(* PLC project MQTT, CODESYS CODESYS V3.5 SP15 Patch 2, author Stefan Dreyer *)
(* stored: creationDateTime 2020-04-11T22:53:20.5572817, version 1.1.0.2, modificationDateTime 2020-04-11T22:45:00.0583058, organization Stefan Dreyer *)
(* MQTT Stuff
Using some cool stuff of OSCAT libs.
see oscat.de

more to describe *)

{attribute 'qualified_only'}
{attribute 'strict'}
TYPE ERRORS : (NOT_VALID := 0, CONNECTION_REFUSED := 1, MAX_PING_REPEATS := 2, RECEIVED_PUBISH_TO_BIG_FOR_BUFFER := 3, FULL_PACKET_NOT_RECEIVED := 4, RECEIVED_PUBLISH_REMAINING_LENGTH_ERROR := 5, NO_MORE_RECEIVE_SLOTS_FREE := 6, CONNECTION_ESTABLISHED := 7, TIMEOUT_CONNECTION := 8, REPEAT_PUBLISH_PUBCOMP := 9, REPEAT_PUBREL := 10, REORDER_PUBREC := 11, REORDER_PUBLISH_OUTGOING := 12, REPEAT_PUBLISH_PUBREC := 13, REPEAT_PUBLISH_PUBACK := 14, HARD_DISCONNECT := 15, MOVED_TO_BIG_RECEIVE_BUFFER := 16, NEED_BUFFER_MOV := 17, UNKNOWN_PAKET_RECEIVED := 18, TO_BIG_PAKET := 19, TOPIC_MOVED_DOWN := 20, TOPIC_AND_PAYLOAD_MOVED := 21, PAYLOAD_MOVED_UP := 22, TOPIC_MOVED_DOWN_NETWORK := 23, PAYLOAD_MOVED_UP_NETWORK := 24, REPEAT_PUBREC := 25, PUBEC_DISCHARGE := 26, REODER_PUBLISH_INCOMMING := 27, REORDER_PUBCOMP := 28, UNKNOWN_PAKET_IN_MQTT_IN_OUT := 29, PUBLISH_NO_SLOT_FREE := 30, OUT_OFF_DYN_MEMORY := 31);
END_TYPE

{attribute 'qualified_only'}
{attribute 'strict'}
TYPE INSERT_SPLIT_RETURN : (INSERT_NOT_VALID := 0, INSERT_DONE, INSERT_PENDING, INSERT_ERROR);
END_TYPE

TYPE MESSAGETYPE : (CONNECT := 16#10, CONNACK := 16#20, PUBLISH := 16#30, PUBACK := 16#40, PUBREC := 16#50, PUBREL := 16#60, PUBCOMP := 16#70, SUBSCRIBE := 16#80, SUBACK := 16#90, UNSUBSCRIBE := 16#A0, UNSUBACK := 16#B0, PINGREQ := 16#C0, PINGRESP := 16#D0, DISCONNECT := 16#E0) BYTE;
END_TYPE

{attribute 'qualified_only'}
{attribute 'strict'}
TYPE PROG_NUM : (Publish, Subscribe, ParseIncomming, MoveBuffer, ParsePublish, GetBufferFreePos, GetSplitTopic, DESTROY_HANDLE_MQTT, DESTROY_SPLIT_TOPIC, STATE_MASHINE_IN, STATE_MASHINE_OUT, SendOutData, SendInData, SendOutDataInsertTopic, SendOutDataInsertPayload, DESTROY_SPLIT_TOPIC_DONE, DESTROY_HANDLE_MQTT_DONE, DESTROY_CALLBACK_COLLECTOR, DESTROY_CALLBACK_COLLECTOR_DONE);
END_TYPE

{attribute 'qualified_only'}
{attribute 'strict'}
TYPE PUSHOVER_SOUND : (Standart := 1);
END_TYPE

TYPE QoS : (AtMostOnce := 2#0, AtLeastOnce := 2#1, ExactlyOnce := 2#10, Fail := 2#10000000) BYTE;
END_TYPE

{attribute 'qualified_only'}
{attribute 'strict'}
TYPE RECEIVE_TYPS : (FIND_PAYLOAD := 0, FIND_TOPIC := 1, FIND_LAST_TOPIC := 2, FIND_LAST_TOPIC_AND_PAYLOAD := 3);
END_TYPE

(* values of RECEIVER_INIT_TYPS: FIND_FULL_TOPIC: searching for full matching topic; FIND_LAST_TOPIC: searching for match of last topic; FIND_PAYLOAD: searching on paylod, from start, spared with delimiter; JSON_FULL: search full topic and one JSON element; JSON_SMALL: searching for last topic and one JSON element; MQTT_STRING: search with MQTT string(including +, #); MQTT_STRING_JSON: search with MQTT string(including +, #), then JSON *)

{attribute 'qualified_only'}
{attribute 'strict'}
TYPE RECEIVER_INIT_TYPS : (FIND_FULL_TOPIC := 0, FIND_LAST_TOPIC, FIND_PAYLOAD, JSON_FULL, JSON_SMALL, MQTT_STRING, MQTT_STRING_JSON);
END_TYPE

{attribute 'qualified_only'}
{attribute 'strict'}
TYPE STEPS_IN : (WAIT_DATA := 0, SEND_PUBACK, SEND_PUBREC, WAIT_PUBREL, SEND_PUBCOMP);
END_TYPE

{attribute 'qualified_only'}
{attribute 'strict'}
TYPE STEPS_OUT : (WAIT_DATA := 0, SEND_PUBLSIH, WAIT_PUBREC, SEND_PUBREL, WAIT_PUBCOMP, WAIT_PUBACK, WAIT_PINGRESP, SEND_SUBSCRIBE, WAIT_SUBACK, SEND_UNSUBSCRIBE, WAIT_UNSUBACK);
END_TYPE

{attribute 'qualified_only'}
{attribute 'strict'}
TYPE TOPIC_MATCH : (TOPIC_MATCHES := 1, TOPIC_DONT_MATCHES := 2, TOPIC_NO_MEMORY := 3) BYTE;
END_TYPE

{attribute 'qualified_only'}
{attribute 'strict'}
TYPE TOPIC_VALID : (TOPIC_UNTESTED := 0, TOPIC_VALID := 2, TOPIC_NOT_VALID := 1, TOPIC_NO_TEST := 3) BYTE;
END_TYPE

(* this data is passed to a subscription callback *)
TYPE CALLBACK_DATA : STRUCT
  PayloadString : POINTER TO STRING(255);  (* the Payload String, be aware, this pointer will only copy 255 bytes. If more needed, use memmove! *)
  Payload : POINTER TO BYTE;  (* pointer to binary payload *)
  PayloadSize : UDINT;  (* size of binary payload *)
  TopicOut : POINTER TO STRING(255);  (* here you get the compleete received topic string, maybe bigger then 255 byte! *)
  TopicOutSplit : POINTER TO SPLIT_TOPIC;  (* split topic.... *)
  PayloadIsString : BOOL;  (* Payload is string *)
END_STRUCT;
END_TYPE

{attribute 'enable_dynamic_creation'}
TYPE CALLBACK_INSTANCES : STRUCT
  callback : MQTT_SUBSCRIBE_CALLBACK;
  next : POINTER TO CALLBACK_INSTANCES := 0;
END_STRUCT;
END_TYPE

TYPE LIST_ALLVALUES_CALLBACK_DATA : STRUCT
  VarTYPE : CommonTypesAndFunctions.VAR_TYPES;
  Target : CommonTypesAndFunctions.ALL_TYPES_UNION_POINTER;
  SubTopic : POINTER TO STRING;  (* pointer to last subtopic or Payload Data to compare with *)
END_STRUCT;
END_TYPE

TYPE LIST_STRING_CALLBACK_DATA : STRUCT
  Target : POINTER TO STRING;  (* pointer to target string *)
  SubTopic : POINTER TO STRING;  (* pointer to last subtopic or Payload Data to compare with *)
END_STRUCT;
END_TYPE

TYPE MQTT_SUBSCRIBE_CALLBACKS : STRUCT
  Callback : MQTT_SUBSCRIBE_CALLBACK;
  ExpectingString : BOOL;  (* expecting string *)
  SplitTopic : POINTER TO HandleSplitTopic;
  free : BOOL := TRUE;  (* set to false if slot is aquired by an subscription *)
END_STRUCT;
END_TYPE

(* here the maximum sizes of paylod and topics are defined if dynamic low init of split topic is used, don't care about MaxTopicElementSize *)
TYPE COM_CONFIG : STRUCT
  MaxPayloadSize : UDINT := 2000;  (* max payload size *)
  MaxTopicLevels : UINT := 25;  (* max topic levels *)
  MaxTopicElementSize : UINT := 255;  (* Max Topic elemt size *)
END_STRUCT;
END_TYPE

TYPE DATA_FROM_BROKER : STRUCT
  MqttTopic : POINTER TO STRING;  (* use array in size of network buffer to split message dynamic, maybe not ... best is dynamic mammory.... or use an array of Pointer.... or callbacks so lets try to buffer public messages and releas one per cycle to application... now we try dynamic memmory.... MQTT Topic from Broker *)
  Topics : POINTER TO SPLIT_TOPIC;
  MqttPayload : POINTER TO BYTE;  (* MQTT Payload for Broker Payload from broker --> Pointer *)
  MqttPayloadSize : UDINT;  (* Payload size *)
  MessageType : MESSAGETYPE;  (* MQTT Message Type *)
  DataReceived : BOOL;  (* Data received *)
END_STRUCT;
END_TYPE

TYPE DATA_TO_BROKER : STRUCT
  PaketData : PAKET_DATA;  (* Data of Paket *)
END_STRUCT;
END_TYPE

(* contro struct between HANDLE_MQTT and MQTT_CONTROL *)
TYPE MQTT_COM : STRUCT
  S_BUF : NETWORK_BUFFER;
  R_BUF : NETWORK_BUFFER;
  MQTT_CON : BOOL;  (* if falling edge close with disconnect packet *)
  MQTT_ABORT : BOOL;  (* if using this to disconnect, don't send disconnect paket.... *)
  MQTT_URL : STRING(OSCAT_BASIC.STRING_LENGTH);
  MQTT_PACKET_NO : WORD;
  TIMEOUT : TIME;
  TLS : BOOL;  (* DNS_IP4 : DWORD; set to true if you want to use TLS *)
  TLS_CONFIG : POINTER TO CommonTypesAndFunctions.TLS_CONFIG := 0;  (* data to TLS stuff *)
  MQTT_RCV_STATE : BYTE;  (* 0= non 1= received 2= error *)
  ERROR_C : DWORD;
  ERROR_T : BYTE;
  CLIENT_ID : STRING(23);  (* CONNECT_TO_LOCALHOST:BOOL; *)
  CLIENT_WILL_TOPIC : STRING(255);  (* Topic vof will message after client id *)
  CLIENT_WILL_MESSAGE_DEAD : STRING(255);
  CLIENT_WILL_RETAIN : BOOL := TRUE;
  MQTT_NO_AWNSER : BOOL;  (* pakte wihout request-- return to receive state 1 *)
END_STRUCT;
END_TYPE

TYPE MQTT_IN_DATA : STRUCT
  step : STEPS_IN;
  PaketID : WORD;
  WaitsForBuffFree : ULINT;
  TimeOut : ton;
  TimeOutStarted : BOOL;
  PUBLISHOrder : UINT;
  PUBCOMPOrder : UINT;
  QoS : QoS;
  CountPubrecRepeat : UINT;
END_STRUCT;
END_TYPE

TYPE MQTT_IN_OUT : STRUCT
  handleFB : POINTER TO HANDLE_MQTT;  (* pointer to handle FB *)
  In : POINTER TO PAKET_DATA;
  InFree : BOOL := TRUE;  (* in free, true if free *)
  TDI : CommonTypesAndFunctions.TIME_DATE_IMPULS_DATA;  (* time, date, impulse... *)
  TLS_CONFIG : POINTER TO CommonTypesAndFunctions.TLS_CONFIG := 0;  (* TLS stuff data *)
  BROKER_CONNECTED : BOOL;
  COM_CONFIG : COM_CONFIG;  (* config for boot up *)
  ClientID : STRING(23) := 'CODESYS_MQTT';  (* client ID, only chars 0123456789abcdefghijklmnopqrstuvwxyzABCDEFGHIJKLMNOPQRSTUVWXYZ" System never can be anonymos *)
  BuildWillTopicAndMessage : BOOL := TRUE;
  WillTopicBase : STRING(255) := 'MQTTWill';
  ClientWillTopic : STRING(255) := 'DEAD';
  ClientWillMessage : STRING(30) := 'DIED';
  dynMemUsage : UDINT;  (* usage of dynamic RAM *)
  disconnectOnBufferOverflow : BOOL;  (* set this to one if you want the client to act like the standardt says if set to one and we receve mor publish pakets than we can handle, QoS 0 packets are lost and QoS 1 and 2 packets have to be repeaded by he broker *)
END_STRUCT;
END_TYPE

TYPE MQTT_INFO : STRUCT
  MQTT_CONNECTED : BOOL;
  MQTT_ERROR : STRING(OSCAT_BASIC.STRING_LENGTH);
END_STRUCT;
END_TYPE

TYPE MQTT_OUT_DATA : STRUCT
  InDataFromFb : POINTER TO PAKET_DATA;
  step : STEPS_OUT;
  WaitsForBuffFree : ULINT;
  PUBRECOrder : UINT;
  TimeOut : ton;
  TimeOutStarted : BOOL;
  PUBLISHOrder : UINT;
  PUBRELRepeatCounter : UINT;
END_STRUCT;
END_TYPE

TYPE ONE_ERROR : STRUCT
  error : ERRORS;
  when : DT;
  ERROR_C : DWORD;
  ERROR_T : BYTE;
  text : STRING(255);
END_STRUCT;
END_TYPE

TYPE PAKET_DATA : STRUCT
  MqttTopic : POINTER TO STRING;  (* MQTT Topic for Broker *)
  MqttTopicLength : UINT;  (* Topic length *)
  MqttPayload : POINTER TO BYTE;  (* MQTT Payload for Broker *)
  MqttPayloadLength : UDINT;  (* Payload length *)
  MessageType : MESSAGETYPE;  (* MQTT Message Type *)
  MessageQoS : QoS;  (* MQTT QoS *)
  SubackQoS : QoS;  (* SUCACK QoS Response *)
  MessageRetain : BOOL;  (* MQTT reatin *)
  DUP : BOOL;  (* Retry of paket *)
  PaketId : WORD;  (* PakatID for header *)
  SendSucsess : BOOL;  (* ID of MQTT FB to store or of request to Broker FbId:UINT; Send was succsessfull *)
  Callback : MQTT_SUBSCRIBE_CALLBACK;  (* Callback FB for subscription *)
  SplitTopic : POINTER TO HandleSplitTopic;  (* split topic for subscribe *)
  CallbackError : BOOL;  (* errore registering the callback *)
  ExpectingString : BOOL;  (* Expecting String *)
END_STRUCT;
END_TYPE

TYPE PUSHOVER_DATA : STRUCT
  Trigger : POINTER TO BOOL;
  Topic : POINTER TO STRING;
  Payload : POINTER TO STRING;
  Prio : USINT;
  Sound : PUSHOVER_SOUND;
  IsConfig : BOOL;
  R_T : R_TRIG;
  NeedToPush : BOOL;
  Negate : BOOL;
END_STRUCT;
END_TYPE

(* used for test cases... *)
TYPE RECEIVE_PAKET : STRUCT
  MqttTopic : STRING(2000);  (* MQTT Topic *)
  MqttPayload : STRING(2000);  (* MQTT Payload *)
END_STRUCT;
END_TYPE

TYPE REMAINING_LENGTH_RETURN : STRUCT
  RemainingLength : UDINT;
  IndexAfterRemainingLength : UINT;
  Error : BOOL;
  BuffToSmall : BOOL;  (* not all bytes of remaining length in buffer... *)
  SizeRemainingLength : USINT;  (* size of remaining length *)
END_STRUCT;
END_TYPE

TYPE SEND_INFOS : STRUCT
  SubscribeIndex : UINT;  (* this index is to be subscribed *)
  SubscribeNeeded : BOOL := FALSE;
  SubscribeBlocking : BOOL;
  UnsubscribeIndex : UINT;  (* this index is to be subscribed *)
  UnsubscribeNeeded : BOOL := FALSE;
  UnsubscribeBlocking : BOOL;
  PublishBlocking : BOOL;  (* this index is to be published *)
  PublishBlockingIndex : UINT;
  PingIndex : UINT;  (* this index is to be published *)
  PingNeeded : BOOL;
END_STRUCT;
END_TYPE

TYPE SPLIT_TOPIC : STRUCT
  Topics : POINTER TO POINTER TO STRING;  (* this is going to be a pointer to a array of pointer to stings *)
  ValidFields : UINT;  (* count of vailid fields in the array *)
END_STRUCT;
END_TYPE

{attribute 'qualified_only'}
VAR_GLOBAL CONSTANT  (* MyConstants *)
  QoS_BUFFER_SIZE : UINT := 50;
  NETWORK_BUFFER_LONG_SIZE : UINT := 4095;
  KEEP_ALIVE_TIME : DWORD := 8;
  SENDING_TIMEOUT : TIME := TIME#4s0ms;
  REPEAT_TIMEOUT : TIME := TIME#2s0ms;
  REORDER_VALUE : UINT := 50000;  (* 50000 *)
  SUBSTRACTION_VALUE : UINT := 30000;  (* 20000 *)
  MAX_PUBREL_REPEATS : UINT := 10;
END_VAR

{attribute 'qualified_only'}
VAR_GLOBAL  (* GVL_MQTT *)
  ProgNum : PROG_NUM;  (* Last Progamm stat for debug timeout exception *)
  LOG_BUFFER_MOVES : BOOL;
END_VAR

INTERFACE MQTT_SUBSCRIBE_CALLBACK
METHOD PublishReceived : BOOL
  VAR_INPUT
    Data : CALLBACK_DATA;  (* Collection of received Data *)
  END_VAR
END_METHOD
END_INTERFACE

PROGRAM Doku

            (*

Hello There,

with this library you are able to send and recvice MQTT paket on all QoS levels 0-2.

Use Pubish to publish data(Strings and binary),

Use subscribe to receive MQTT data. On Subscribe you can tell the FB if you are expecting an String as data, so you will get one on the pointer output.

How to use you can see in the example and testCase FB. This is my Test Case an it does up to 100 send and receives per second on an raspberry PI 1+ connectet to an mosquitto broker on an 
windows 10 maschine.

If you find errors, or anny instability, tell me, i will have a look.

TLS works fine without certificates.

This Projekt i using some parts of the grat OSCAT libs, so take a look at oscat.de

Greatings 

*)
          
END_PROGRAM

FUNCTION_BLOCK TestOutOfTheBoxNoTLS
  VAR_INPUT
    client : STRING := 'test.mosquitto.org:1883';  (* test.mosquitto.org *)
  END_VAR
  VAR
    MQTTClient : HANDLE_MQTT;
    MQTT_IN_OUT : MQTT_IN_OUT;
    publish : MQTTPublish;
    subscribe : MQTTSubscribe;
    ReceiveSubscribeTopic : STRING(255);
    ReceiveSubscribePayloadTick : STRING(255);
    ReceiveSubscribePayloadState : STRING(255);
    State : MQTTState;
    init : BOOL;
    varSend : BOOL;
    timerSend : ton;
    t1 : ton;
    t2 : ton;
    Payload : STRING;
    StringCallback : ListStringCallback;  (* the method PublishReceved() is call when an publsih packet form the broker is received. *)
    CallBackTargets : ARRAY[0..1] OF LIST_STRING_CALLBACK_DATA := [(Target := ADR(ReceiveSubscribePayloadState), SubTopic := ADR('State')), (Target := ADR(ReceiveSubscribePayloadTick), SubTopic := ADR('Tick'))];  (* the array contains the targets and sub topics for receive *)
  END_VAR

            //here init is done
IF NOT init THEN
	init := TRUE;
	MQTT_IN_OUT.ClientID := CONCAT('CodesysMqtt',TO_STRING(TICKS.GetTick(xDummy:= TRUE)));
	publish.SetMqttInOut(MQTT_IN_OUT:= ADR(MQTT_IN_OUT));
	subscribe.SetMqttInOut(MQTT_IN_OUT:= ADR(MQTT_IN_OUT));
	//init state FB, so you only have to call state();without parameters... 
	State.Init(
	State:= ADR(t1.Q), 
	Topic:= ADR('CODESYS-MQTT-BY-SD/State'), 
	StateName:= ADR(''), 
	StateValueOn:= ADR('On'), 
	StateValueOff:= ADR('Off'), 
	QoS:= QoS.ExactlyOnce, 
	RetainMqtt:= TRUE,
	MQTT_IN_OUT:= ADR(MQTT_IN_OUT));
	StringCallback.InitAsSplitTopic(ListData := ADR(CallBackTargets), LengthOfData:= 2);

END_IF
//timer for repeating packets
timerSend(in := NOT varSend, PT := T#2S);
varSend := timerSend.Q; 
t1(IN:= NOT t2.Q, PT:= T#1S, );
t2(IN:= t1.Q, PT:= T#1S, );
//call of MQTT client
MQTTClient( 
	MQTT_IN_OUT:= MQTT_IN_OUT, 
	ENABLE:= TRUE, 
	URL:= client, 
	TIMEOUT:= T#5S, 
	TLS:= FALSE);
//build payload
IF varSend THEN
	Payload:= TO_STRING(TICKS.GetTick(xDummy:= TRUE));
END_IF
//Publish Payload
publish(
	Topic:= ADR('CODESYS-MQTT-BY-SD/Tick'), 
	PayloadString:= ADR(Payload), 
	PublishAsString:= TRUE, 
	QoSIn:= QoS.ExactlyOnce, 
	MRetain:= TRUE, 
	send:= varSend);
//Subscribe to topic
subscribe(
	Subscribe:= TRUE, 
	Topic:= ADR('CODESYS-MQTT-BY-SD/#'), 
	QoSSubscribe:= QoS.ExactlyOnce, 
	ExpectingString:= TRUE,
	Callback:= StringCallback);


//call of state FB
State();
          
END_FUNCTION_BLOCK

FUNCTION_BLOCK TestOutOfTheBoxTLS
  VAR_INPUT
    client : STRING := 'test.mosquitto.org:8883';  (* test.mosquitto.org *)
  END_VAR
  VAR
    MQTTClient : HANDLE_MQTT;
    MQTT_IN_OUT : MQTT_IN_OUT;
    publish : MQTTPublish;
    subscribe : MQTTSubscribe;
    ReceiveSubscribeTopic : STRING(255);
    ReceiveSubscribePayloadTick : STRING(255);
    ReceiveSubscribePayloadState : STRING(255);
    State : MQTTState;
    init : BOOL;
    varSend : BOOL;
    timerSend : ton;
    t1 : ton;
    t2 : ton;
    Payload : STRING;
    StringCallback : ListStringCallback;  (* the method PublishReceved() is call when an publsih packet form the broker is received. *)
    CallBackTargets : ARRAY[0..1] OF LIST_STRING_CALLBACK_DATA := [(Target := ADR(ReceiveSubscribePayloadState), SubTopic := ADR('State')), (Target := ADR(ReceiveSubscribePayloadTick), SubTopic := ADR('Tick'))];  (* the array contains the targets and sub topics for receive *)
    TLS_CONFIG : CommonTypesAndFunctions.TLS_CONFIG;
  END_VAR

            //here init is done
IF NOT init THEN
	init := TRUE;
	MQTT_IN_OUT.ClientID := CONCAT('CodesysMqtt',TO_STRING(TICKS.GetTick(xDummy:= TRUE)));
	publish.SetMqttInOut(MQTT_IN_OUT:= ADR(MQTT_IN_OUT));
	subscribe.SetMqttInOut(MQTT_IN_OUT:= ADR(MQTT_IN_OUT));
	//init state FB, so you only have to call state();without parameters... 
	State.Init(
	State:= ADR(t1.Q), 
	Topic:= ADR('CODESYS-MQTT-BY-SD/State'), 
	StateName:= ADR(''), 
	StateValueOn:= ADR('On'), 
	StateValueOff:= ADR('Off'), 
	QoS:= QoS.ExactlyOnce, 
	RetainMqtt:= TRUE,
	MQTT_IN_OUT:= ADR(MQTT_IN_OUT));
	StringCallback.InitAsSplitTopic(ListData := ADR(CallBackTargets), LengthOfData:= 2);
	MQTT_IN_OUT.TLS_CONFIG := ADR(TLS_CONFIG);
END_IF
//timer for repeating packets
timerSend(in := NOT varSend, PT := T#2S);
varSend := timerSend.Q; 
t1(IN:= NOT t2.Q, PT:= T#1S, );
t2(IN:= t1.Q, PT:= T#1S, );
//call of MQTT client
MQTTClient( 
	MQTT_IN_OUT:= MQTT_IN_OUT, 
	ENABLE:= TRUE, 
	URL:= client, 
	TIMEOUT:= T#5S, 
	TLS:= TRUE);
//build payload
IF varSend THEN
	Payload:= TO_STRING(TICKS.GetTick(xDummy:= TRUE));
END_IF
//Publish Payload
publish(
	Topic:= ADR('CODESYS-MQTT-BY-SD/Tick'), 
	PayloadString:= ADR(Payload), 
	PublishAsString:= TRUE, 
	QoSIn:= QoS.ExactlyOnce, 
	MRetain:= TRUE, 
	send:= varSend);
//Subscribe to topic	
subscribe(
	Subscribe:= TRUE, 
	Topic:= ADR('CODESYS-MQTT-BY-SD/#'), 
	QoSSubscribe:= QoS.ExactlyOnce, 
	ExpectingString:= TRUE,
	Callback:= StringCallback);


//call of state FB
State();
          
END_FUNCTION_BLOCK

(* true if levels the same *)
FUNCTION CheckTopicLevel : BOOL
  VAR_INPUT
    s1 : POINTER TO STRING;  (* String from Broker *)
    s2 : POINTER TO STRING;  (* Subscribe String *)
  END_VAR
  VAR
    LenS1 : UINT;
  END_VAR

            CheckTopicLevel := FALSE;
//test Wildcard
IF (s2^[0] = CommonTypesAndFunctions.GetChar(in:= '+')) THEN //(s2[0] = GetChar(in:= '#')) OR  don't check # here
	CheckTopicLevel := TRUE;
	RETURN;	
END_IF
LenS1 := CommonTypesAndFunctions.len(STR:= s1); 
IF (LenS1 <> CommonTypesAndFunctions.len(STR:= s2)) THEN 
	RETURN;
END_IF//if len not eval then return
IF (CommonTypesAndFunctions.find(STR1:= s1, STR2:= s2) >= 0) OR (LenS1 = 0)THEN
	CheckTopicLevel := TRUE;
END_IF
          
END_FUNCTION

FUNCTION DoRemainingLength : USINT
  VAR_INPUT
    buffer : POINTER TO BYTE;
    RemainingLength : UINT;
  END_VAR
  VAR
    LocalLength : LINT;
    LocalBuffer : ARRAY[0..3] OF BYTE;
    BufferIndex : UINT := 0;
    TmpByte : BYTE;
  END_VAR

            //check if we have to move data for inserting remaining length
//borders are given in the mqtt doku
//
IF RemainingLength <= 128 THEN
	buffer[1] := UINT_TO_BYTE(RemainingLength);
	DoRemainingLength := 0;
ELSE
	LocalLength := RemainingLength;
	REPEAT
		TmpByte := LINT_TO_BYTE(LocalLength MOD 128);
		LocalLength := LocalLength / 128;
		IF LocalLength > 0 THEN
			TmpByte := TmpByte OR 128;
		END_IF
		LocalBuffer[BufferIndex] := TmpByte; 
		BufferIndex := BufferIndex +1;
	UNTIL 
		LocalLength <= 0 
	END_REPEAT
	//now move mem	
	//buffer index points to NEXT field, so sub 1
	MEM.MemMove(pSource:= buffer+2, pDestination:= buffer + 2 + BufferIndex - 1 , uiNumberOfBytes:= RemainingLength);
	CASE BufferIndex OF
		2: 	buffer[1]:= LocalBuffer[0];
			buffer[2]:= LocalBuffer[1];
			DoRemainingLength := 1;
		3:	buffer[1]:= LocalBuffer[0];
			buffer[2]:= LocalBuffer[1];
			buffer[3]:= LocalBuffer[2];
			DoRemainingLength := 2;
		4:	buffer[1]:= LocalBuffer[0];
			buffer[2]:= LocalBuffer[1];
			buffer[3]:= LocalBuffer[2];
			buffer[4]:= LocalBuffer[3];
			DoRemainingLength := 3;
		
	END_CASE
	
END_IF

          
END_FUNCTION

(* here no move of data, call remainig length bevor moving topic and paylod, use this for borders are given in the mqtt doku use this for publish pakets *)
FUNCTION DoRemainingLengthBevor : USINT
  VAR_INPUT
    buffer : POINTER TO BYTE;  (* points to start of buffer, not to start of remainig length! *)
    SizeTopic : UDINT;
    SizePayload : UDINT;
    InQoS : QoS;
  END_VAR
  VAR
    RemainingLength : UDINT;
    LocalLength : LINT;
    LocalBuffer : ARRAY[0..3] OF BYTE;
    BufferIndex : UINT := 0;
    TmpByte : BYTE;
  END_VAR

            
	
RemainingLength := SizeTopic + SizePayload;
	
RemainingLength := RemainingLength + 2;//add topic size encoding space
IF NOT (InQoS = QoS.AtMostOnce) THEN
	RemainingLength := RemainingLength + 2;//add space for paket identifier
END_IF

IF RemainingLength <= 128 THEN
	buffer[1] := UDINT_TO_BYTE(RemainingLength);
	DoRemainingLengthBevor := 0;
ELSE
	LocalLength := RemainingLength;
	REPEAT
		TmpByte := LINT_TO_BYTE(LocalLength MOD 128);
		LocalLength := LocalLength / 128;
		IF LocalLength > 0 THEN
			TmpByte := TmpByte OR 128;
		END_IF
		LocalBuffer[BufferIndex] := TmpByte; 
		BufferIndex := BufferIndex +1;
	UNTIL 
		LocalLength <= 0 
	END_REPEAT
	CASE BufferIndex OF
		2: 	buffer[1]:= LocalBuffer[0];
			buffer[2]:= LocalBuffer[1];
			DoRemainingLengthBevor := 1;
		3:	buffer[1]:= LocalBuffer[0];
			buffer[2]:= LocalBuffer[1];
			buffer[3]:= LocalBuffer[2];
			DoRemainingLengthBevor := 2;
		4:	buffer[1]:= LocalBuffer[0];
			buffer[2]:= LocalBuffer[1];
			buffer[3]:= LocalBuffer[2];
			buffer[4]:= LocalBuffer[3];
			DoRemainingLengthBevor := 3;
		
	END_CASE
	
END_IF

          
END_FUNCTION

FUNCTION GetRemainingLength : REMAINING_LENGTH_RETURN
  VAR_INPUT
    Buff : POINTER TO BYTE;  (* Pointer to Buffer *)
    pos : UINT;  (* Start of data in Buffer *)
    BuffSize : UDINT;
  END_VAR
  VAR
    BufferIndex : UINT := 1;
    Multipler : UDINT := 1;
    TmpByte : BYTE;
  END_VAR

            GetRemainingLength.Error := FALSE;
GetRemainingLength.SizeRemainingLength:= 0;

GetRemainingLength.BuffToSmall := FALSE;
BufferIndex := pos + 1;
REPEAT
	IF BufferIndex > (BuffSize - 1) THEN
		GetRemainingLength.BuffToSmall := TRUE;
	ELSE
		TmpByte := Buff[BufferIndex];
		BufferIndex := BufferIndex + 1;
		GetRemainingLength.RemainingLength := GetRemainingLength.RemainingLength + (TmpByte AND 127) * Multipler;
		Multipler := Multipler *128;
		IF Multipler > 128*128*128 THEN
			GetRemainingLength.RemainingLength := 0;//lengt 0 if broken
			GetRemainingLength.Error := TRUE;
		END_IF
	END_IF
	GetRemainingLength.SizeRemainingLength := GetRemainingLength.SizeRemainingLength + 1;
UNTIL
	TmpByte.7 = FALSE OR GetRemainingLength.BuffToSmall
	//TmpByte.7 = FALSE  OR GetRemainingLength.RemainingLength = 0 OR GetRemainingLength.BuffToSmall
END_REPEAT
GetRemainingLength.IndexAfterRemainingLength := BufferIndex;
          
END_FUNCTION

FUNCTION InitMQTTValue : BOOL
  VAR_INPUT
    DataArray : POINTER TO CommonTypesAndFunctions.PWConfigs;
    CountOfArray : UINT;
    ValueToMQTTArray : POINTER TO MQTTValue;
    MQTT_IN_OUT : POINTER TO MQTT_IN_OUT;
  END_VAR
  VAR
    i : UINT;
  END_VAR

            FOR i := 0 TO CountOfArray - 1 DO
	IF DataArray[i].NeedsMQTT THEN
		ValueToMQTTArray[i].Init(
			Topic:= DataArray[i].MQTTTopic, 
			ValueName:= DataArray[i].MQTTName, 
			ValuePointer:= DataArray[i].PointerTo, 
			ValueType:= DataArray[i].ValueType, 
			ValueDiff:= DataArray[i].MQTTDiff, 
			DecimalPlace:= DataArray[i].MQTTDezimal, 
			QoS:= DataArray[i].MQTTQoS, 
			RetainMqtt:= DataArray[i].MQTTRetain, 
			MinTime:= DataArray[i].MQTTTime,
			MQTT_IN_OUT:= MQTT_IN_OUT);
	END_IF
END_FOR
          
END_FUNCTION

(* returnds new pos in buff *)
FUNCTION InsertStringToBufferAndLength : UINT
  VAR_INPUT
    Str : POINTER TO STRING;
    buff : POINTER TO BYTE;  (* address to buffer *)
    pos : UINT;  (* Start to insert *)
  END_VAR
  VAR
    length : UINT;
  END_VAR

            length := CommonTypesAndFunctions.LEN(Str);
buff[pos]:= OSCAT_BASIC.BYTE_OF_DWORD(in:= length, N:= 1);
buff[pos+1]:= OSCAT_BASIC.BYTE_OF_DWORD(in:= length, N:= 0);

MEM.MemMove(pSource:= str, pDestination:= ADR(buff[pos+2]), uiNumberOfBytes:= length);
InsertStringToBufferAndLength := pos + length + 2;
          
END_FUNCTION

(* this FB collects instances of FB with the MQTT_SUBSCRIBE_CALLBACK interface. then you can pass a instance of this FB to a subscription FB to call all of your FBs to a specific subscription topic, in this call you can check if the packet was for your instance. If your instance methode call return true, the the FB exits the loop an so you may save cycle time. MEmory for instance references are created dynamic, so no restriction by library *)
FUNCTION_BLOCK CallbackCollector IMPLEMENTS MQTT_SUBSCRIBE_CALLBACK
  VAR
    first : POINTER TO CALLBACK_INSTANCES := 0;
    items : UDINT;
    size : UDINT;
  END_VAR

            
          

(* true if all ok, else false *)
METHOD put : BOOL
  VAR_INPUT
    instance : MQTT_SUBSCRIBE_CALLBACK;
  END_VAR
  VAR
    aktElement : POINTER TO CALLBACK_INSTANCES;
  END_VAR
                  aktElement := first;

IF aktElement = 0 THEN
	//first hit...
	{info 'semaphore'}
	first := __NEW(CALLBACK_INSTANCES);
	IF first = 0 THEN
		put := FALSE;
		RETURN;
	END_IF
	aktElement := first;
ELSE
	//search last
	WHILE aktElement^.next  <> 0 DO 
		aktElement := aktElement^.next; 
	END_WHILE
	{info 'semaphore'}
	aktElement^.next := __NEW(CALLBACK_INSTANCES);
	IF aktElement^.next = 0 THEN
		put := FALSE;
		RETURN;
	END_IF
	aktElement := aktElement^.next;
END_IF

aktElement^.callback := instance;
put := TRUE;
items := items + 1;
size := size + SIZEOF(CALLBACK_INSTANCES);
                
END_METHOD

METHOD PublishReceived : BOOL
  VAR_INPUT
    Data : CALLBACK_DATA;  (* Collection of received Data *)
  END_VAR
  VAR
    element : POINTER TO CALLBACK_INSTANCES;
    loop : BOOL := TRUE;
  END_VAR
                  

IF first = 0 THEN
	//no callback avalable
	RETURN;
END_IF
element := first;


WHILE loop DO
	IF element^.callback.PublishReceived(Data := Data) THEN
		PublishReceived := TRUE;
		RETURN;
	END_IF
	IF element^.next = 0 THEN
		loop := FALSE;
	ELSE
		element := element^.next;
	END_IF
END_WHILE

                
END_METHOD

(* destroy all dynamic content *)
METHOD destroy : BOOL
  VAR
    aktElement : POINTER TO CALLBACK_INSTANCES;
    nextElement : POINTER TO CALLBACK_INSTANCES;
  END_VAR
                  GVL_MQTT.ProgNum := PROG_NUM.DESTROY_CALLBACK_COLLECTOR;
IF first = 0 THEN
	RETURN;
END_IF

aktElement := first;

REPEAT
	nextElement := aktElement^.next;
	__DELETE(aktElement);
	aktElement := nextElement;
	items := items - 1;
	size := size - SIZEOF(CALLBACK_INSTANCES);
UNTIL aktElement = 0
END_REPEAT
first := 0;
GVL_MQTT.ProgNum := PROG_NUM.DESTROY_CALLBACK_COLLECTOR_DONE;
                
END_METHOD

METHOD FB_Exit : BOOL
  VAR_INPUT
    bInCopyCode : BOOL;  (* TRUE: the exit method is called in order to leave the instance which will be copied afterwards (online change). *)
  END_VAR
                  destroy();
                
END_METHOD
END_FUNCTION_BLOCK

FUNCTION_BLOCK ReceiverBase
  VAR
    MatchTyp : RECEIVER_INIT_TYPS;
    Target : CommonTypesAndFunctions.ALL_TYPES_UNION_POINTER;
    TargetType : CommonTypesAndFunctions.VAR_TYPES;
    PayloadCompare : POINTER TO STRING;
    TopicCompare : POINTER TO STRING;
    delimiter : BYTE;
    delimiterString : STRING(3);
    SplitTopic : HandleSplitTopic;
  END_VAR

            
          

METHOD init
  VAR_INPUT
    MQTT_IN_OUT : POINTER TO MQTT_IN_OUT;
    MatchTyp : RECEIVER_INIT_TYPS;
    Target : CommonTypesAndFunctions.ALL_TYPES_UNION_POINTER;
    TargetType : CommonTypesAndFunctions.VAR_TYPES;
    PayloadCompare : POINTER TO STRING;
    TopicCompare : POINTER TO STRING;
    delimiter : BYTE;
  END_VAR
                  MatchTyp := MatchTyp;
Target := Target;
TargetType := TargetType;
PayloadCompare := PayloadCompare;
TopicCompare := TopicCompare;
delimiter := delimiter;
delimiterString[0] := delimiter;
delimiterString[1] := 0;

IF MatchTyp = RECEIVER_INIT_TYPS.MQTT_STRING or MatchTyp = RECEIVER_INIT_TYPS.MQTT_STRING_JSON THEN
	SplitTopic.LowInit(TopicsLevelInit:= MQTT_IN_OUT^.COM_CONFIG.MaxTopicLevels,
			 SplitElementSizeInit:= MQTT_IN_OUT^.COM_CONFIG.MaxTopicElementSize, dynMemUsageInit:= ADR(MQTT_IN_OUT^.dynMemUsage));
	SplitTopic.NewTopic(in:= TopicCompare, test:= TRUE, SizeOfString:= CommonTypesAndFunctions.len(str:= TopicCompare));
END_IF
                
END_METHOD

METHOD CheckMatch : BOOL
  VAR_INPUT
    Data : CALLBACK_DATA;  (* Collection of received Data *)
  END_VAR
  VAR
    foundPos : DINT;
  END_VAR
                  CheckMatch := FALSE;
CASE MatchTyp OF
	RECEIVER_INIT_TYPS.FIND_FULL_TOPIC:
		IF CommonTypesAndFunctions.StrEquals(str1:= Data.TopicOut , str2:= PayloadCompare) THEN
			CheckMatch := TRUE;
			GetValue(fromWhere:= Data.PayloadString);
			RETURN;
		END_IF 
	RECEIVER_INIT_TYPS.FIND_LAST_TOPIC:
		IF CommonTypesAndFunctions.StrEquals(str1:= Data.TopicOutSplit^.Topics[Data.TopicOutSplit^.ValidFields - 1], str2:= PayloadCompare) THEN
			CheckMatch := TRUE;
			GetValue(fromWhere:= Data.PayloadString);
			RETURN;
		END_IF
	RECEIVER_INIT_TYPS.FIND_PAYLOAD:
		IF CommonTypesAndFunctions.StrEqualsAtStartWithDelimiter(str1:= PayloadCompare, str2:= Data.PayloadString , delimiter:= delimiter) THEN
			CheckMatch := TRUE;
			GetValue(fromWhere:= Data.PayloadString + TO_UINT(CommonTypesAndFunctions.find(str1:= Data.PayloadString, str2:= ADR(delimiterString)))+1);
			RETURN;	
		END_IF
	RECEIVER_INIT_TYPS.JSON_FULL:
		IF CommonTypesAndFunctions.StrEquals(str1:= Data.TopicOut , str2:= PayloadCompare) THEN
			foundPos := CommonTypesAndFunctions.find(str1:= Data.PayloadString, str2:= TopicCompare); 
			IF foundPos >= 0 THEN
				CheckMatch := TRUE;
				RETURN;	
			END_IF
		END_IF
	RECEIVER_INIT_TYPS.JSON_SMALL:
		IF CommonTypesAndFunctions.StrEquals(str1:= Data.TopicOutSplit^.Topics[Data.TopicOutSplit^.ValidFields - 1], str2:= PayloadCompare) THEN
			IF CommonTypesAndFunctions.find(str1:= Data.PayloadString, str2:= TopicCompare) >= 0 THEN
				CheckMatch := TRUE;
				RETURN;	
			END_IF
		END_IF
	RECEIVER_INIT_TYPS.MQTT_STRING:
		IF SplitTopic.CheckTopicMatchToMe(with:= Data.TopicOutSplit) = TOPIC_MATCH.TOPIC_MATCHES THEN
			CheckMatch := TRUE;
			RETURN;
		END_IF
	RECEIVER_INIT_TYPS.MQTT_STRING_JSON:
		IF SplitTopic.CheckTopicMatchToMe(with:= Data.TopicOutSplit) = TOPIC_MATCH.TOPIC_MATCHES THEN
			IF CommonTypesAndFunctions.find(str1:= Data.PayloadString, str2:= TopicCompare) >= 0 THEN
				CheckMatch := TRUE;
				RETURN;	
			END_IF
		END_IF
	
END_CASE
                
END_METHOD

METHOD GetValue
  VAR_INPUT
    fromWhere : POINTER TO STRING(65000);
  END_VAR
                  CASE TargetType OF
	CommonTypesAndFunctions.VAR_TYPES.BOOL_T,
	CommonTypesAndFunctions.VAR_TYPES.BYTE_T,
	CommonTypesAndFunctions.VAR_TYPES.DATE_T,
	CommonTypesAndFunctions.VAR_TYPES.DINT_T,
	CommonTypesAndFunctions.VAR_TYPES.DT_T,
	CommonTypesAndFunctions.VAR_TYPES.DWORD_T,
	CommonTypesAndFunctions.VAR_TYPES.INT_T,
	CommonTypesAndFunctions.VAR_TYPES.LINT_T,
	CommonTypesAndFunctions.VAR_TYPES.LREAL_T,
	CommonTypesAndFunctions.VAR_TYPES.LWORD_T,
	CommonTypesAndFunctions.VAR_TYPES.REAL_T,
	CommonTypesAndFunctions.VAR_TYPES.SINT_T,
	CommonTypesAndFunctions.VAR_TYPES.TIME_T,
	CommonTypesAndFunctions.VAR_TYPES.TOD_T,
	CommonTypesAndFunctions.VAR_TYPES.TOD2_T,
	CommonTypesAndFunctions.VAR_TYPES.UDINT_T,
	CommonTypesAndFunctions.VAR_TYPES.UINT_T,
	CommonTypesAndFunctions.VAR_TYPES.ULINT_T,
	CommonTypesAndFunctions.VAR_TYPES.USINT_T,
	CommonTypesAndFunctions.VAR_TYPES.WORD_T:
	CommonTypesAndFunctions.GetValueFromStringPt
				(TypeOfValue:= TargetType, Target:= Target, str:= fromWhere);
END_CASE
                
END_METHOD
END_FUNCTION_BLOCK

FUNCTION_BLOCK ReceiveString IMPLEMENTS MQTT_SUBSCRIBE_CALLBACK
  VAR_OUTPUT
    MQTTReceived : STRING(255);  (* your desired payload... *)
  END_VAR
  VAR
    splitTopic : BOOL;  (* if set to true we search the instance name in the lowest topic *)
    splitPayload : BOOL;  (* if set to true we search the instance name in Payload separatet by the split char *)
    SplitPayloadChar : BYTE;  (* an this is the split char... *)
    MyCompString : POINTER TO STRING;  (* compare with this... *)
    MyReturnHit : BOOL;  (* if set to true and hit we will return true, else false... *)
  END_VAR

            
          

METHOD PublishReceived : BOOL
  VAR_INPUT
    Data : CALLBACK_DATA;  (* Collection of received Data *)
  END_VAR
  VAR
    StrPt : POINTER TO STRING(255);
  END_VAR
                  // no we can check if the topic/payload matches to my compare string 

//now search the right topic 
IF splitTopic THEN
	
	IF CommonTypesAndFunctions.StrEquals(str1:= Data.TopicOut, str2:= MyCompString) THEN
		StrPt := Data.PayloadString;
		MQTTReceived := StrPt^;
		PublishReceived := MyReturnHit;
	END_IF

END_IF

//now look into the payload
IF splitPayload THEN
	
	IF CommonTypesAndFunctions.StrEqualsAtStartWithDelimiter(str1:= MyCompString, str2:= Data.PayloadString, delimiter:= SplitPayloadChar) THEN
		//now search split char
		StrPt := Data.PayloadString;
		StrPt := StrPt + TO_DWORD(CommonTypesAndFunctions.find(str1 := StrPt, str2:= ADR(SplitPayloadChar))) + 1;
		MQTTReceived := StrPt^;
		PublishReceived := MyReturnHit;
	END_IF
END_IF

                
END_METHOD

METHOD initAsFindTopic : BOOL
  VAR_INPUT
    compString : POINTER TO STRING;  (* this i'm searching *)
    returnHit : BOOL;  (* if set to true and hit we will return true, else false... *)
  END_VAR
                  
splitPayload := FALSE;
splitTopic := TRUE;
MyCompString := compString;
MyReturnHit := returnHit;
                
END_METHOD

METHOD initAsFindPayload : BOOL
  VAR_INPUT
    splitChar : STRING;  (* only first char is selected *)
    compString : POINTER TO STRING;  (* this i'm searching *)
    returnHit : BOOL;  (* if set to true and hit we will return true, else false... *)
  END_VAR
                  
splitPayload := TRUE;
splitTopic := FALSE;

SplitPayloadChar := CommonTypesAndFunctions.GetChar(in:= splitChar);
MyCompString := compString;
MyReturnHit := returnHit;
                
END_METHOD
END_FUNCTION_BLOCK

(* Receives one value from a MQTT publish packet. It can check diffrent sources to determinate if the data is for this Value.... *)
FUNCTION_BLOCK ReceiveValue IMPLEMENTS MQTT_SUBSCRIBE_CALLBACK
  VAR_OUTPUT
    MQTTReceived : CommonTypesAndFunctions.ALL_TYPES_UNION;  (* your desired payload... *)
  END_VAR
  VAR
    TargetPointer : CommonTypesAndFunctions.ALL_TYPES_UNION_POINTER;  (* pointer to target *)
    MyValueTyp : CommonTypesAndFunctions.VAR_TYPES;  (* Target var type *)
    SplitPayloadChar : BYTE;  (* an this is the split char... *)
    MyCompString : POINTER TO STRING;  (* compare with this... *)
    MyCompStringPayload : POINTER TO STRING;  (* and this for Payload *)
    MyReturnHit : BOOL;  (* if set to true and hit we will return true, else false... *)
    ReceiveType : RECEIVE_TYPS;
  END_VAR

            
          

METHOD PublishReceived : BOOL
  VAR_INPUT
    Data : CALLBACK_DATA;  (* Collection of received Data *)
  END_VAR
  VAR
    StrPt : POINTER TO STRING;
  END_VAR
                  CASE ReceiveType OF
	RECEIVE_TYPS.FIND_LAST_TOPIC:	
		//now search the right topic 
		IF CommonTypesAndFunctions.StrEquals(str1:= Data.TopicOutSplit^.Topics[Data.TopicOutSplit^.ValidFields - 1], str2:= MyCompString) THEN
			CommonTypesAndFunctions.GetValueFromStringPt(TypeOfValue:= MyValueTyp ,Target:= TargetPointer, str:= DATA.PayloadString);
			PublishReceived := MyReturnHit;
		END_IF
	RECEIVE_TYPS.FIND_PAYLOAD:
		IF CommonTypesAndFunctions.StrEqualsAtStartWithDelimiter(str1:= MyCompString, str2:= Data.PayloadString, delimiter:= SplitPayloadChar) THEN
			//now search split char
			StrPt := Data.PayloadString;
			StrPt := StrPt + TO_DWORD(CommonTypesAndFunctions.find(str1 := StrPt, str2:= ADR(SplitPayloadChar))) + 1;
			CommonTypesAndFunctions.GetValueFromStringPt(TypeOfValue:= MyValueTyp ,Target:= TargetPointer, str:= StrPt);
			PublishReceived := MyReturnHit;
		END_IF
	RECEIVE_TYPS.FIND_LAST_TOPIC_AND_PAYLOAD:
		//now search the right topic and payload
		IF CommonTypesAndFunctions.StrEquals(str1:= Data.TopicOut, str2:= MyCompString) THEN
			IF CommonTypesAndFunctions.StrEqualsAtStartWithDelimiter(str1:= MyCompStringPayload, str2:= Data.PayloadString, delimiter:= SplitPayloadChar) THEN
				StrPt := Data.PayloadString;
				StrPt := StrPt + TO_DWORD(CommonTypesAndFunctions.find(str1 := StrPt, str2:= ADR(SplitPayloadChar))) + 1;
				CommonTypesAndFunctions.GetValueFromStringPt(TypeOfValue:= MyValueTyp ,Target:= TargetPointer, str:= StrPt);
				PublishReceived := MyReturnHit;
			END_IF
		END_IF
	RECEIVE_TYPS.FIND_TOPIC:
		//now search the right topic 
		IF CommonTypesAndFunctions.StrEquals(str1:= Data.TopicOut, str2:= MyCompString) THEN
			CommonTypesAndFunctions.GetValueFromStringPt(TypeOfValue:= MyValueTyp ,Target:= TargetPointer, str:= DATA.PayloadString);
			PublishReceived := MyReturnHit;
		END_IF
END_CASE


                
END_METHOD

METHOD initAsFindPayload : BOOL
  VAR_INPUT
    splitChar : STRING;  (* only first char is selected *)
    compString : POINTER TO STRING;  (* this i'm searching *)
    ValueTyp : CommonTypesAndFunctions.VAR_TYPES;  (* this typ is my received string *)
    returnHit : BOOL;  (* if set to true and hit we will return true, else false... *)
  END_VAR
                  ReceiveType := RECEIVE_TYPS.FIND_PAYLOAD;

SplitPayloadChar := CommonTypesAndFunctions.GetChar(in:= splitChar);
MyCompString := compString;
MyValueTyp := ValueTyp;
makePointer();
MyReturnHit := returnHit;
                
END_METHOD

(* this will only check the lowest topic level *)
METHOD initAsFindTopic : BOOL
  VAR_INPUT
    compString : POINTER TO STRING;  (* this i'm searching *)
    ValueTyp : CommonTypesAndFunctions.VAR_TYPES;  (* this typ is my received string *)
    returnHit : BOOL;  (* if set to true and hit we will return true, else false... *)
  END_VAR
                  ReceiveType := RECEIVE_TYPS.FIND_TOPIC;
MyCompString := compString;
MyValueTyp := ValueTyp;
makePointer();
MyReturnHit := returnHit;
                
END_METHOD

METHOD makePointer : BOOL
                  TargetPointer := CommonTypesAndFunctions.MakeAllTypesPointer(fromWho:= adr(MQTTReceived), myType:= MyValueTyp);
                
END_METHOD

(* this will check the whole topic! *)
METHOD initAsFindTopicAndPayload : BOOL
  VAR_INPUT
    splitChar : STRING;  (* only first char is selected *)
    compStringTopic : POINTER TO STRING;  (* this topic i'm searching *)
    compStringPayload : POINTER TO STRING;  (* this payload i'm searching *)
    ValueTyp : CommonTypesAndFunctions.VAR_TYPES;  (* this typ is my received string *)
    returnHit : BOOL;  (* if set to true and hit we will return true, else false... *)
  END_VAR
                  ReceiveType := RECEIVE_TYPS.FIND_LAST_TOPIC_AND_PAYLOAD;
SplitPayloadChar := CommonTypesAndFunctions.GetChar(in:= splitChar);
MyCompString := compStringTopic;
MyCompStringPayload := compStringPayload;
MyValueTyp := ValueTyp;
makePointer();
MyReturnHit := returnHit;
                
END_METHOD

METHOD SetOutput : BOOL
  VAR_INPUT
    value : CommonTypesAndFunctions.ALL_TYPES_UNION;
  END_VAR
                  MQTTReceived := value;
                
END_METHOD

METHOD initAsFindLastTopic : BOOL
  VAR_INPUT
    compString : POINTER TO STRING;  (* this i'm searching *)
    ValueTyp : CommonTypesAndFunctions.VAR_TYPES;  (* this typ is my received string *)
    returnHit : BOOL;  (* if set to true and hit we will return true, else false... *)
  END_VAR
                  ReceiveType := RECEIVE_TYPS.FIND_LAST_TOPIC;
MyCompString := compString;
MyValueTyp := ValueTyp;
makePointer();
MyReturnHit := returnHit;
                
END_METHOD
END_FUNCTION_BLOCK

FUNCTION_BLOCK ReceiveValueWithStrucur EXTENDS ReceiveValue
  VAR
    InstanceName : CommonTypesAndFunctions.GetInstanceName;
    localCompString : STRING(255);
  END_VAR

            


          

METHOD InitReceiveStructur : BOOL
  VAR_INPUT
    TopicLevel : USINT;
    ValueTyp : CommonTypesAndFunctions.VAR_TYPES;  (* this typ is my received string *)
    returnHit : BOOL;  (* if set to true and hit we will return true, else false... *)
  END_VAR
  VAR
    tString : STRING(255);
    cmpByte : BYTE;
    bytePointer : POINTER TO BYTE;
    StringPointer : POINTER TO STRING;
    i : UINT;
  END_VAR
                  
tString:= InstanceName.GetInstanceTopic();

cmpByte:= CommonTypesAndFunctions.GetChar('/');

bytePointer := ADR(tString) + CommonTypesAndFunctions.len(ADR(tString));

i := 0;

WHILE bytePointer >= ADR(tString) DO
	IF bytePointer^ = cmpByte THEN
		i := i + 1; 
	END_IF
	
	IF i = TopicLevel THEN
		
		StringPointer := bytePointer + 1;
		//ReceiveTopic := GVL_ZIGBEE.TextZigbeeTopic;
		//ReceiveTopic := CONCAT(STR1:= ReceiveTopic, STR2:= StringPointer^); 
		localCompString := StringPointer^;
		initAsFindTopic(compString:= ADR(localCompString), ValueTyp:= ValueTyp, returnHit:= returnHit);
		RETURN;
	END_IF
	bytePointer := bytePointer - 1;
END_WHILE
localCompString := tString;
initAsFindTopic(compString:= ADR(localCompString), ValueTyp:= ValueTyp, returnHit:= returnHit);
                
END_METHOD
END_FUNCTION_BLOCK

(* this FB expects all values as a string, binary receive is not suported... Payload content is only value, no description, no special characters... *)
FUNCTION_BLOCK ListAllValuesCallback IMPLEMENTS MQTT_SUBSCRIBE_CALLBACK
  VAR
    MyListData : POINTER TO LIST_ALLVALUES_CALLBACK_DATA;
    MyLengthOfData : ULINT;
    ListSplitTopic : BOOL;
    ListSplitPayload : BOOL;
    SplitCharPayload : BYTE;
  END_VAR

            
          

METHOD PublishReceived : BOOL
  VAR_INPUT
    Data : CALLBACK_DATA;  (* Collection of received Data *)
  END_VAR
  VAR
    i : ULINT;
    StrPt : POINTER TO STRING;
  END_VAR
                  IF ListSplitTopic THEN
	//now search the right topic 
	FOR i := 0 TO MyLengthOfData - 1 DO
		IF CommonTypesAndFunctions.StrEquals(str1:= Data.TopicOutSplit^.Topics[Data.TopicOutSplit^.ValidFields - 1], str2:= MyListData[i].SubTopic) THEN
			CommonTypesAndFunctions.GetValueFromStringPt(TypeOfValue:= MyListData[i].VarTYPE ,Target:= MyListData[i].Target, str:= DATA.PayloadString);
		END_IF
	END_FOR
END_IF
IF ListSplitPayload THEN
	FOR i := 0 TO MyLengthOfData - 1 DO
		IF CommonTypesAndFunctions.StrEqualsAtStartWithDelimiter(str1:= MyListData[i].SubTopic, str2:= Data.PayloadString, delimiter:= SplitCharPayload) THEN
			//now search split char
			StrPt := Data.PayloadString;
			StrPt := StrPt + TO_DWORD(CommonTypesAndFunctions.find(str1 := StrPt, str2:= ADR(SplitCharPayload))) + 1;
			
			CommonTypesAndFunctions.GetValueFromStringPt(TypeOfValue:= MyListData[i].VarTYPE ,Target:= MyListData[i].Target, str:= StrPt);
		END_IF
	END_FOR
	
END_IF
                
END_METHOD

METHOD InitAsSplitTopic : BOOL
  VAR_INPUT
    Data : POINTER TO LIST_ALLVALUES_CALLBACK_DATA;
    LengthOfData : ULINT;  (* Count of List Data *)
  END_VAR
                  MyListData := Data;
MyLengthOfData := LengthOfData;
ListSplitTopic := TRUE;
ListSplitPayload := FALSE;
                
END_METHOD

(* inits FB, callback methoth then checks if the payload ist the same in the first characters as in the template make sure to receive a string payload! *)
METHOD InitAsSplitPayload : BOOL
  VAR_INPUT
    Data : POINTER TO LIST_ALLVALUES_CALLBACK_DATA;
    LengthOfData : ULINT;  (* Count of List Data *)
    SplitChar : BYTE;  (* spliting character *)
  END_VAR
                  MyListData :=Data;
MyLengthOfData := LengthOfData;
ListSplitTopic := FALSE;
ListSplitPayload := TRUE;
SplitCharPayload := SplitChar;
                
END_METHOD
END_FUNCTION_BLOCK

FUNCTION_BLOCK ListStringCallback IMPLEMENTS MQTT_SUBSCRIBE_CALLBACK
  VAR
    MyListData : POINTER TO LIST_STRING_CALLBACK_DATA;
    MyLengthOfData : ULINT;
    ListSplitTopic : BOOL;
    ListSplitPayload : BOOL;
    SplitCharPayload : BYTE;
  END_VAR

            
          

METHOD PublishReceived : BOOL
  VAR_INPUT
    Data : CALLBACK_DATA;  (* Collection of received Data *)
  END_VAR
  VAR
    i : ULINT;
    StrPt : POINTER TO STRING(255);
    SplitPos : DINT;
  END_VAR
                  //now search the right topic 
IF ListSplitTopic THEN
	FOR i := 0 TO MyLengthOfData - 1 DO
		IF CommonTypesAndFunctions.StrEquals(str1:= Data.TopicOutSplit^.Topics[Data.TopicOutSplit^.ValidFields - 1], str2:= MyListData[i].SubTopic) THEN
			//MyListData[i].Target^ := Data.PayloadString^;
			MEM.MemMove(pSource:= Data.PayloadString, pDestination:= MyListData[i].Target, uiNumberOfBytes:= TO_UINT(data.PayloadSize + 1));
			PublishReceived := TRUE;
		END_IF
	END_FOR
END_IF

IF ListSplitPayload THEN
	FOR i := 0 TO MyLengthOfData - 1 DO
		IF CommonTypesAndFunctions.StrEqualsAtStartWithDelimiter(str1:= MyListData[i].SubTopic, str2:= Data.PayloadString, delimiter:= SplitCharPayload) THEN
			//now search split char
			StrPt := Data.PayloadString;
			SplitPos := CommonTypesAndFunctions.find(str1 := StrPt, str2:= ADR(SplitCharPayload));
			StrPt := StrPt + TO_DWORD(SplitPos) + 1;
			//MyListData[i].Target^ := StrPt^;
			MEM.MemMove(pSource:= Data.PayloadString, pDestination:= MyListData[i].Target, uiNumberOfBytes:= TO_UINT(data.PayloadSize + 1 - TO_UDINT(SplitPos)) );
			PublishReceived := TRUE;
		END_IF
	END_FOR
	
END_IF

                
END_METHOD

(* ints FB to split packets at lowest payload level *)
METHOD InitAsSplitTopic : BOOL
  VAR_INPUT
    ListData : POINTER TO LIST_STRING_CALLBACK_DATA;
    LengthOfData : ULINT;  (* Count of List Data *)
  END_VAR
                  MyListData :=ListData;
MyLengthOfData := LengthOfData;
ListSplitTopic := TRUE;
ListSplitPayload := FALSE;

                
END_METHOD

(* inits FB, callback methoth then checks if the payload ist the same in the first characters as in the template make sure to receive a string payload! *)
METHOD InitAsSplitPayload : BOOL
  VAR_INPUT
    ListData : POINTER TO LIST_STRING_CALLBACK_DATA;
    LengthOfData : ULINT;  (* Count of List Data *)
    SplitChar : BYTE;  (* spliting character *)
  END_VAR
                  MyListData :=ListData;
MyLengthOfData := LengthOfData;
ListSplitTopic := FALSE;
ListSplitPayload := TRUE;
SplitCharPayload := SplitChar;
                
END_METHOD
END_FUNCTION_BLOCK

(* this FB expects all values as a string, binary receive is not suported... Payload content is only value, no description, no special characters... *)
FUNCTION_BLOCK AllValuesCallback IMPLEMENTS MQTT_SUBSCRIBE_CALLBACK
  VAR_OUTPUT
    received : BOOL;  (* data was received, you have to reset this bit after checking! *)
  END_VAR
  VAR
    VarType : CommonTypesAndFunctions.VAR_TYPES;
    MyTarget : CommonTypesAndFunctions.ALL_TYPES_UNION_POINTER;
  END_VAR

            
          

METHOD PublishReceived : BOOL
  VAR_INPUT
    Data : CALLBACK_DATA;  (* Collection of received Data *)
  END_VAR
                  CommonTypesAndFunctions.GetValueFromStringPt(TypeOfValue:= VarType,Target:= MyTarget, str:= DATA.PayloadString);

received := TRUE;
                
END_METHOD

METHOD Init : BOOL
  VAR_INPUT
    SetType : CommonTypesAndFunctions.VAR_TYPES;
    Target : CommonTypesAndFunctions.ALL_TYPES_UNION_POINTER;
  END_VAR
                  VarType := SetType;
MyTarget := Target;

                
END_METHOD

METHOD ResetReceived : BOOL
                  received := FALSE;

                
END_METHOD
END_FUNCTION_BLOCK

FUNCTION_BLOCK SingelStringCallback IMPLEMENTS MQTT_SUBSCRIBE_CALLBACK
  VAR_OUTPUT
    received : BOOL;  (* data was received, you have to reset this bit after checking! *)
  END_VAR
  VAR
    MyPayload : POINTER TO STRING;
    MyTopic : POINTER TO STRING;
  END_VAR

            
          

METHOD PublishReceived : BOOL
  VAR_INPUT
    Data : CALLBACK_DATA;  (* Collection of received Data *)
  END_VAR
                  MEM.MemMove(pSource:= Data.PayloadString, pDestination:= MyPayload, uiNumberOfBytes:= TO_UINT(data.PayloadSize + 1));
MEM.MemMove(pSource:= Data.TopicOut, pDestination:= MyTopic, uiNumberOfBytes:= CommonTypesAndFunctions.len(Data.TopicOut) + 1);

received := TRUE;
                
END_METHOD

METHOD Init : BOOL
  VAR_INPUT
    payload : POINTER TO STRING;
    topic : POINTER TO STRING;
  END_VAR
                  MyTopic := topic;
MyPayload := payload;
                
END_METHOD

METHOD ResetReceived : BOOL
                  received := FALSE;

                
END_METHOD
END_FUNCTION_BLOCK

(* var/log/mosquitto/mosquitto.log Messsages are not beeing repeatet, if timout for an answer then connection is canceled, new established and the publisher have to start new Start the command line subscriber: mosquitto_sub -v -t 'test/topic' mosquitto_sub -v -h test.mosquitto.org -t 'test/topic' sudo apt-get install tshark tshark -i 1 -a duration:60 -w /tmp/wlan.pcap debug / logging : mosquitto_sub -v -t '$SYS/#' sudo nano /etc/mosquitto/mosquitto.conf --> 'log_type all' Publish test message with the command line publisher: mosquitto_pub -t 'test/topic' -m 'helloWorld' change check free to InFbNo kopieren sudo cp /var/log/mosquitto/mosquitto.log /tmp/ zugriff sudo chmod -v a=r /tmp/mosquitto.log TODO: Take care of clean session, is enabled, do it paramable? *)
FUNCTION_BLOCK HANDLE_MQTT
  VAR_IN_OUT
    MQTT_IN_OUT : MQTT_IN_OUT;
  END_VAR
  VAR_INPUT
    ENABLE : BOOL;
    URL : STRING(OSCAT_BASIC.STRING_LENGTH);  (* use format: user:password@domain:port *)
    TIMEOUT : TIME;
    TLS : BOOL;
  END_VAR
  VAR_OUTPUT
    ERROR_C : DWORD;
    ERROR_T : BYTE;
  END_VAR
  VAR
    MQTT_INFO : MQTT_INFO;
    DT_MQTT : CommonTypesAndFunctions.TIME_DATE_IMPULS;
    MQTT_CONTROL : MQTT_CONTROL;
    step : INT;
    i1 : UINT;
    PingSlot : UINT;
    COM : MQTT_COM;
    connected : BOOL;
    TimeoutConnection : TON;
    MqttsDoneIo : ULINT;
    CycleTime : DWORD;
    LastCycleTime : DWORD;
    NextPingTime : CAA.TICK;
    PingTime : CAA.TICK := ((MyConstants.KEEP_ALIVE_TIME * 1000) - 6000);  (* next ping after 6 seconds *)
    PingRequestet : BOOL;  (* Ping was sendet *)
    PingData : DATA_TO_BROKER;
    myFbNo : UINT;
    PubrelOrderIndexCounter : UINT;
    PubcompOrderIndexCounter : UINT;
    LogFile : CAA.HANDLE;  (* log file *)
    open : FILE.Open;
    write : FILE.Write;
    LogString : STRING(255);
    DebugFile : BOOL := FALSE;
    OutData : ARRAY[0..MyConstants.QoS_BUFFER_SIZE] OF MQTT_OUT_DATA;
    InData : ARRAY[0..MyConstants.QoS_BUFFER_SIZE] OF MQTT_IN_DATA;
    PublishSendListCount : UINT;
    PublishSendList : ARRAY[0..MyConstants.QoS_BUFFER_SIZE] OF UINT;
    PubrelSendListCount : UINT;
    PubrelSendList : ARRAY[0..MyConstants.QoS_BUFFER_SIZE] OF UINT;
    PubackSendListCount : UINT;
    PubackSendList : ARRAY[0..MyConstants.QoS_BUFFER_SIZE] OF UINT;
    PubrecSendListCount : UINT;
    PubrecSendList : ARRAY[0..MyConstants.QoS_BUFFER_SIZE] OF UINT;
    PubcompSendListCount : UINT;
    PubcompSendList : ARRAY[0..MyConstants.QoS_BUFFER_SIZE] OF UINT;
    RepeatedPublish : ULINT;  (* Repeted Publishs *)
    RepeatedPublishsAfterPubrel : ULINT;  (* Repeatet publishs afert ot much repeat of pubrel *)
    RepeatedPubrel : ULINT;  (* Repeted pubrel *)
    CountRepeatedPing : ULINT;  (* Repeted Ping *)
    CountRepeatedPingDisconnect : UINT;  (* Repeated pings untill disconnect *)
    PublishsUnacknowledged : UINT;  (* count of Publishs unacknowledged *)
    LastToBigTopic : STRING(255);  (* last part of 255 chars of to big paket topic *)
    CountToBigTopics : ULINT;  (* count of to big topics *)
    CountLengthErrors : ULINT;  (* Cont of ength Error Pakets *)
    CountRepeatPublishReceive : ULINT;  (* Count of repeatet publishs *)
    CountReceivedPublishs : ULINT;  (* Count Received Publishs *)
    CountSendedPublishs : ULINT;  (* count sended publishs *)
    CountRepeatSubscribe : ULINT;  (* Count of repeated subscribs *)
    CountRepeatUnsubscribe : ULINT;  (* Count of repeated unsubscribs *)
    CountRepeatetPubrec : ULINT;  (* Count of repeatet pubrec *)
    CountOutputPublishCalled : ULINT;  (* Count of OutputPublish calls *)
    PUBREC_ERROR_ID_BUFFER : ARRAY[0..(PUBREC_ERROR_ID_BUFFER_SIZE - 1)] OF UINT;
    PUBREC_ERROR_INDEX : UINT;
    OutgoingPublishOrderIndexCounter : UINT;  (* send Publish order Index *)
    IncomingPublishOrderIndexCounter : UINT;  (* receive Publish order Index *)
    CountReceivePubrelUnknown : ULINT;  (* Received Pubrel, Paket not found *)
    CountReceiveUnsubackUnknown : ULINT;  (* Received Unsuback, Paket not found *)
    CountReceiveSubackUnknown : ULINT;  (* Received Suback, Paket not found *)
    CountReceivePubackUnknown : ULINT;  (* Received Puback, Paket not found *)
    CountReceivePubrecUnknown : ULINT;  (* Received Pubrec, Paket not found *)
    CountReceivePubcompUnknown : ULINT;  (* Received Pubcomp, Paket not found *)
    SendInfos : SEND_INFOS;
    CountOutSendNotFree : ULINT;
    CountInSendNotFree : ULINT;
    CountCantSendPublishBufferToFull : ULINT;
    CounterPublishSendForMonitor : UINT;
    PublishsSendPerSeconde : UINT;
    CounterPublishReceivedForMonitor : UINT;
    PublishsReceivedPerSeconde : UINT;
    NotKnownPaket : MESSAGETYPE;
    CountUnkownPaket : ULINT;
    LastPaktetForUnkownPaket : MESSAGETYPE;
    HelperLastPaktetForUnkownPaket : MESSAGETYPE;
    CountBufferMoves : ULINT;
    CountNothingSend : ULINT;
    CountConnectAttempt : ULINT;
    CountSplitTopicSizeExceeded : ULINT;  (* count of topic size exceeded *)
    CountWaitForRestOfPaket : ULINT;
    CountResetBufferIn : ULINT;
    InBufferMoved : UINT;
    SendFree : BOOL;
    MySplitTopic : HandleSplitTopic;
    InsertSplitTopic : InsertSplitTopic;
    InsertSplitPayload : InsertSplitPayload;
    StepBuildPublish : INT;
    StepBuildSubscribe : INT;
    StepBuildUnsubscribe : INT;
    SplitPublishBuffer : POINTER TO BYTE;  (* use this buffer for received publish packets whos size exceded network buffer Size *)
    SplitPublishBufferSize : UDINT;
    SplitPublishLength : UDINT;
    MaxPublishPacketSize : UDINT;  (* output from buffer Don't write new data! SplitPublishLock:BOOL; *)
    PayloadMemorySize : DWORD;
    SubscribeCallbacks : ARRAY[0..(CALLBACKS_BUFFER_SIZE - 1)] OF MQTT_SUBSCRIBE_CALLBACKS;
    TopicMemorySize : DWORD;
    COM_CONFIG : COM_CONFIG;
    PublishSplited : BOOL;  (* publish paket broken, waiting for more data *)
    DoDisconnect : BOOL;
    SendetBytes : ULINT;
    ReceivedBytes : ULINT;
    InSlotsWorking : UINT;
    OutSlotsWorking : UINT;
    SplitPublishBufferAllocationSize : UDINT;
    DynMemUsagePointer : POINTER TO UDINT;
    CallbacksFull : BOOL;  (* callbacks array full *)
    ErrorHistory : ARRAY[0..COUNT_ERROR_HISTORY] OF ONE_ERROR;
    localTdi : CommonTypesAndFunctions.TIME_DATE_IMPULS_DATA;
    StepInitDone : BOOL;  (* Step 10 Init is done: *)
  END_VAR
  VAR CONSTANT
    CALLBACKS_BUFFER_SIZE : UINT := 200;
    RECEIVE_PUBLISH_BUFFER_SIZE : UINT := (NETWORK_BUFFER_LONG_SIZE * 2);
    TRANSMIT_BUFFER_SIZE : UINT := NETWORK_BUFFER_LONG_SIZE;
    SIZE_PUBREL : UINT := 4;
    SIZE_UNSUBACK : UINT := 4;
    SIZE_PINGRESP : UINT := 2;
    SIZE_PINGREQ : UINT := 2;
    SIZE_SUBACK : UINT := 5;
    SIZE_PUBACK : UINT := 4;
    SIZE_PUBREC : UINT := 4;
    SIZE_PUBCOMP : UINT := 4;
    SIZE_PAKET_BUFFER_HEADER : UINT := 4;
    PUBREC_ERROR_ID_BUFFER_SIZE : UINT := 100;
    MAX_PING_REPEATS : UINT := 10;
    SPLIT_PUBLISH_BUFFER_ADDITIONAL_RAM : UINT := 17;
    COUNT_MAX_PUBREC_REPEAT_TO_DISCHARGE : UINT := 20;
    COUNT_ERROR_HISTORY : UINT := 1000;
  END_VAR

            IF MQTT_INFO.MQTT_CONNECTED THEN
	SendFree := COM.S_BUF.SIZE = 0;	
END_IF

CycleTime := OSCAT_BASIC.T_PLC_MS() - LastCycleTime;
LastCycleTime := OSCAT_BASIC.T_PLC_MS();
//get system time and so one
DT_MQTT(
	TDI_Data:= MQTT_IN_OUT.TDI);
localTdi:= MQTT_IN_OUT.TDI ; 
TimeoutConnection(IN:= step = 10, PT:= T#5S);

IF DebugFile THEN
		//open log file
		open(
	xExecute:= TRUE, 
	sFileName:= '/tmp/mqtt.log', 
	eFileMode:= 0, 
	xExclusive:= TRUE, 
	hFile=> LogFile);
END_IF

CASE step OF

	00:	MQTT_IN_OUT.BROKER_CONNECTED := FALSE;
		IF ENABLE THEN
			MQTT_IN_OUT.handleFB := THIS;
			PingRequestet := FALSE;
			PublishsUnacknowledged := 0;
			PUBREC_ERROR_INDEX := 0;
			CountRepeatedPingDisconnect := 0;
			SendetBytes := 0;
			ReceivedBytes := 0;		
			PublishSplited := FALSE;
			DoDisconnect := FALSE;
			SendInfos.PingNeeded := FALSE;
			SendInfos.SubscribeNeeded := FALSE;
			SendInfos.UnsubscribeNeeded := FALSE;
			StepBuildPublish := 0;
			StepBuildSubscribe := 0;
			StepBuildUnsubscribe := 0;
			InsertSplitTopic.reset();
			InsertSplitPayload.reset();
			CountConnectAttempt := CountConnectAttempt + 1;
			DynMemUsagePointer := ADR(MQTT_IN_OUT.dynMemUsage);
			COM.MQTT_URL := URL;
			COM.TIMEOUT := TIMEOUT;
			COM.CLIENT_ID := MQTT_IN_OUT.ClientID;
			COM.TLS := TLS;
			COM.TLS_CONFIG := MQTT_IN_OUT.TLS_CONFIG;
			ResetPingTime();
			//build will topic
			IF MQTT_IN_OUT.BuildWillTopicAndMessage THEN
				COM.CLIENT_WILL_TOPIC := MQTT_IN_OUT.WillTopicBase;
				COM.CLIENT_WILL_TOPIC := Standard.CONCAT(STR1:= COM.CLIENT_WILL_TOPIC, '/');
				COM.CLIENT_WILL_TOPIC := Standard.CONCAT(STR1:= COM.CLIENT_WILL_TOPIC, STR2:= COM.CLIENT_ID);
				COM.CLIENT_WILL_TOPIC := Standard.CONCAT(STR1:= COM.CLIENT_WILL_TOPIC, '/');
				COM.CLIENT_WILL_TOPIC := Standard.CONCAT(STR1:= COM.CLIENT_WILL_TOPIC, MQTT_IN_OUT.ClientWillTopic);
				COM.CLIENT_WILL_TOPIC := Standard.CONCAT(STR1:= '/', COM.CLIENT_WILL_TOPIC);
				COM.CLIENT_WILL_TOPIC := Standard.CONCAT(STR1:= COM.CLIENT_ID, COM.CLIENT_WILL_TOPIC);
			ELSE
				COM.CLIENT_WILL_TOPIC := MQTT_IN_OUT.ClientWillTopic;
			END_IF
			COM.CLIENT_WILL_MESSAGE_DEAD := MQTT_IN_OUT.ClientWillMessage;
			COM_CONFIG := MQTT_IN_OUT.COM_CONFIG;
			FOR i1 := 0 TO MyConstants.QoS_BUFFER_SIZE - 1 DO
				//reset in slots
				InData[i1].step := STEPS_IN.WAIT_DATA;
				OutData[i1].step := STEPS_OUT.WAIT_DATA;
				//reset Timeouts...
				InData[i1].TimeOutStarted := FALSE;
				OutData[i1].TimeOutStarted := FALSE;
				InData[i1].TimeOut(IN:= InData[i1].TimeOutStarted, PT:= MyConstants.REPEAT_TIMEOUT);
				OutData[i1].TimeOut(IN:= OutData[i1].TimeOutStarted, PT:= MyConstants.REPEAT_TIMEOUT);
			END_FOR
			//reset callbacks
			FOR i1 := 0 TO CALLBACKS_BUFFER_SIZE - 1 DO
				SubscribeCallbacks[i1].free := TRUE; 
			END_FOR
			IF  MySplitTopic.FullInit(TopicsLevelInit:= COM_CONFIG.MaxTopicLevels, SplitElementSizeInit:= COM_CONFIG.MaxTopicElementSize, dynMemUsageInit:= ADR(MQTT_IN_OUT.dynMemUsage)) THEN
				
				PayloadMemorySize := COM_CONFIG.MaxPayloadSize;
				{warning disable C0033}
				TopicMemorySize := COM_CONFIG.MaxTopicElementSize * COM_CONFIG.MaxTopicLevels;
				MaxPublishPacketSize := (COM_CONFIG.MaxTopicElementSize * COM_CONFIG.MaxTopicLevels) + PayloadMemorySize;
				SplitPublishBufferAllocationSize := MaxPublishPacketSize + SPLIT_PUBLISH_BUFFER_ADDITIONAL_RAM;
				{info 'semaphore'}
				SplitPublishBuffer  := __NEW(BYTE, SplitPublishBufferAllocationSize);//some additional bytes for paket overhead and termination
				IF SplitPublishBuffer = 0 THEN
					PushError(newError:= ERRORS.OUT_OFF_DYN_MEMORY, text:='No Dyn Memory in Step 00 in Handle' );
					step := 60;
				ELSE
					MQTT_IN_OUT.dynMemUsage := MQTT_IN_OUT.dynMemUsage + SplitPublishBufferAllocationSize;
					{warning restore C0033}
		
					step := 10;
					COM.MQTT_CON := TRUE;
					StepInitDone := TRUE;
					
				END_IF
			ELSE
				PushError(newError:= ERRORS.OUT_OFF_DYN_MEMORY, text:='No Dyn Memory in Step 00 in Handle on create SplitTopic' );
				step := 60;
			END_IF
		END_IF	
	10:	IF MQTT_INFO.MQTT_CONNECTED THEN
			step := 40;
			MQTT_IN_OUT.BROKER_CONNECTED := TRUE;
			PushError(newError:= ERRORS.CONNECTION_ESTABLISHED, text:='');
		END_IF
		IF TimeoutConnection.Q THEN
			PushError(newError:= ERRORS.TIMEOUT_CONNECTION, text:='' );
			step := 0;//reset steps
			destroy();
			
		END_IF
	40:	
		IF PublishSplited THEN
			MergeSplitedPublish(MQTT_IN_OUT:= ADR(MQTT_IN_OUT));
		END_IF	
		ParseIncoming(MQTT_IN_OUT:= ADR(MQTT_IN_OUT));
		PublishSendListCount := 0;
		PubrelSendListCount := 0;
		PubackSendListCount := 0;
		PubrecSendListCount := 0;
		PubcompSendListCount := 0;
		StateMashineIn(MQTT_IN_OUT:= ADR(MQTT_IN_OUT));
		StateMashineOut( MQTT_IN_OUT:= ADR(MQTT_IN_OUT));
		
		SendOutData(MQTT_IN_OUT:= ADR(MQTT_IN_OUT));
		SendInData(MQTT_IN_OUT:= ADR(MQTT_IN_OUT));
	
		IF MQTT_IN_OUT.TDI.IMP THEN
			PublishsSendPerSeconde := CounterPublishSendForMonitor;
			CounterPublishSendForMonitor := 0;
			PublishsReceivedPerSeconde := CounterPublishReceivedForMonitor;
			CounterPublishReceivedForMonitor := 0;
		END_IF
		IF COM.S_BUF.SIZE = 0 THEN
			CountNothingSend := CountNothingSend + 1;
		END_IF
		IF NOT ENABLE THEN 	(* beenden? *)
			step := 50;
			
		END_IF;
		IF DoDisconnect THEN
			DoDisconnect := FALSE;
			//here hard disconnect
			PushError(newError:= ERRORS.HARD_DISCONNECT , text:='');
			COM.MQTT_CON := FALSE; (* MQTT Verbindung beenden *)
			COM.MQTT_ABORT := TRUE;
			MQTT_IN_OUT.BROKER_CONNECTED := FALSE;
			step := 60;
		END_IF

(* ~~~~~~~~~~~~~~~~~~~~~~ *)

50: 
	COM.MQTT_CON := FALSE; (* MQTT Verbindung beenden *)
	MQTT_IN_OUT.BROKER_CONNECTED := FALSE;
	step := 60;//wait for disconnect
60:
	IF MQTT_INFO.MQTT_CONNECTED = FALSE THEN
		destroy();
		step := 0;
		MQTT_IN_OUT.BROKER_CONNECTED := FALSE;
	END_IF
END_CASE;



(* ########################## *)

IF CountRepeatedPingDisconnect > MAX_PING_REPEATS THEN
	DoDisconnect := TRUE;
	IF step = 40 THEN
		PushError(newError:= ERRORS.MAX_PING_REPEATS, text:='');
	END_IF
END_IF


SendetBytes := SendetBytes + COM.S_BUF.SIZE;
MQTT_CONTROL(COM:= COM, INFO:=MQTT_INFO);
ReceivedBytes := ReceivedBytes + COM.R_BUF.SIZE;
ERROR_C := COM.ERROR_C;
ERROR_T := COM.ERROR_T;
//handl ping telegram
IF NextPingTime < TICKS.GetTick(xDummy:= TRUE) AND NOT PingRequestet AND connected THEN
	
	MakePingPaket(MQTT_IN_OUT := MQTT_IN_OUT);
	
END_IF

IF COM.ERROR_T > BYTE#0 THEN  (* FEHLER *)
	DoDisconnect := TRUE;
	MQTT_IN_OUT.BROKER_CONNECTED := FALSE;
	PushError(newError:= ERRORS.CONNECTION_REFUSED, text:='');
END_IF;
//put status to local clients
 

connected := MQTT_IN_OUT.BROKER_CONNECTED;
(* ########################## *)

(* revision history


*)
          

METHOD ResetPingTime
                  NextPingTime := PingTime + TICKS.GetTick(xDummy:= TRUE);
CountRepeatedPingDisconnect := 0;
                
END_METHOD

METHOD MakePingPaket
  VAR_IN_OUT
    MQTT_IN_OUT : MQTT_IN_OUT;
  END_VAR
                  IF MQTT_IN_OUT.InFree THEN 
	MQTT_IN_OUT.IN := ADR(PingData); //set request
	PingData.PaketData.MessageType := MESSAGETYPE.PINGREQ;
	MQTT_IN_OUT.InFree := FALSE;
	PingRequestet := TRUE;
END_IF

                
END_METHOD

METHOD StateMashineOut
  VAR_INPUT
    MQTT_IN_OUT : POINTER TO MQTT_IN_OUT;  (* StepData:POINTER TO MQTT_OUT_DATA; *)
  END_VAR
  VAR
    i : UINT;
    j : UINT;
    tmpLowest : UINT;
    minIndex : UINT;
    UnsubscribeLastHighest : UINT := 16#FFFF;
    SubscribeLastHighest : UINT := 16#FFFF;
    ReceivePaketID : WORD;  (* PublishLastHighest : UINT := 16#FFFF; PubrelLastHighest : UINT := 16#FFFF; *)
    ReceivePakteType : BYTE;
    TempSlotsWorking : UINT;
  END_VAR
                  (*need a token for coordinate send of pakets....
prio for Awnser and repeat pakets bevor new publish
dont use token, just send paket with next publish index*)
//get paket id
ReceivePaketID := DWORD_TO_WORD(OSCAT_BASIC.DWORD_OF_BYTE(B3:= 0, B2:= 0, B1:= COM.R_BUF.BUFFER[2], B0:= COM.R_BUF.BUFFER[3]));
ReceivePakteType := COM.R_BUF.BUFFER[0] AND 16#F0; 

GVL_MQTT.ProgNum := PROG_NUM.STATE_MASHINE_OUT;
PublishSendListCount := 0;
PubrelSendListCount := 0;

TempSlotsWorking := 0;
FOR i := 0 TO MyConstants.QoS_BUFFER_SIZE - 1 DO
	//do Timers...
	OutData[i].TimeOut(IN:= OutData[i].TimeOutStarted, PT:= MyConstants.REPEAT_TIMEOUT);
	CASE OutData[i].step OF
		
		STEPS_OUT.WAIT_DATA:
			OutData[i].TimeOutStarted := FALSE;
			IF NOT MQTT_IN_OUT^.InFree THEN//new Data from FBs
				MQTT_IN_OUT^.InFree := TRUE;
				OutData[i].InDataFromFb := MQTT_IN_OUT^.In;//set Data
				//Pakte id = slot + 1....
				OutData[i].InDataFromFb^.PaketId := i + 1;
				CASE OutData[i].InDataFromFb^.MessageType OF
					MESSAGETYPE.PINGREQ:
						OutData[i].step := STEPS_OUT.WAIT_PINGRESP;
						SendInfos.PingNeeded := TRUE;
						SendInfos.PingIndex := i;
						PingSlot := i;
					//we only sending one subscription per subscribe paket....
					MESSAGETYPE.SUBSCRIBE:
						//check if we have a slot free for subscription
						FOR j := 0 TO CALLBACKS_BUFFER_SIZE - 1 DO
							IF SubscribeCallbacks[j].free THEN
								OutData[i].step := STEPS_OUT.SEND_SUBSCRIBE;
								CallbacksFull := FALSE;
								EXIT;
							END_IF
						END_FOR
						IF j = CALLBACKS_BUFFER_SIZE THEN
							//no free slot
							MQTT_IN_OUT^.In^.CallbackError := TRUE;
							CallbacksFull := TRUE;
						END_IF
					MESSAGETYPE.UNSUBSCRIBE:
						OutData[i].step := STEPS_OUT.SEND_UNSUBSCRIBE;
					ELSE
						PushError(newError:= ERRORS.UNKNOWN_PAKET_IN_MQTT_IN_OUT , text:= CONCAT(STR1:= 'Type:', STR2:= TO_STRING(OutData[i].InDataFromFb^.MessageType)));
				END_CASE
				
			END_IF
		
		STEPS_OUT.WAIT_PINGRESP:
			IF OutData[i].TimeOutStarted AND OutData[i].TimeOut.Q AND NOT SendInfos.PingNeeded THEN
				//timeout, need repead
				SendInfos.PingNeeded := TRUE;
				SendInfos.PingIndex := i;
				CountRepeatedPing := CountRepeatedPing + 1; 
				CountRepeatedPingDisconnect := CountRepeatedPingDisconnect + 1;
				OutData[i].TimeOutStarted := FALSE;
			END_IF
		STEPS_OUT.SEND_UNSUBSCRIBE:
			//check if my paket ID is the lowest to send it
			IF OutData[i].InDataFromFb^.PaketId < UnsubscribeLastHighest AND NOT SendInfos.UnsubscribeNeeded THEN
				SendInfos.UnsubscribeIndex := i;
				SendInfos.UnsubscribeNeeded := TRUE;
				UnsubscribeLastHighest := OutData[i].InDataFromFb^.PaketId;
			END_IF	
		STEPS_OUT.WAIT_UNSUBACK:
			IF OutData[i].TimeOutStarted AND OutData[i].TimeOut.Q THEN
				//timeout, need repead
				OutData[i].step := STEPS_OUT.SEND_UNSUBSCRIBE;//repeat subscribe
				CountRepeatUnsubscribe := CountRepeatUnsubscribe + 1;
				OutData[i].TimeOutStarted := FALSE;
			END_IF
		STEPS_OUT.SEND_SUBSCRIBE:
			//check if my paket ID is the lowest to send it
			IF OutData[i].InDataFromFb^.PaketId < SubscribeLastHighest AND NOT SendInfos.SubscribeNeeded THEN
				SendInfos.SubscribeIndex := i;
				SendInfos.SubscribeNeeded := TRUE;
				SubscribeLastHighest := OutData[i].InDataFromFb^.PaketId;
			END_IF	
		STEPS_OUT.WAIT_SUBACK:
			IF OutData[i].TimeOutStarted AND OutData[i].TimeOut.Q THEN
				//timeout, need repead
				OutData[i].step := STEPS_OUT.SEND_SUBSCRIBE;//repeat subscribe
				CountRepeatSubscribe := CountRepeatSubscribe + 1;
				OutData[i].TimeOutStarted := FALSE;
			END_IF
			
		STEPS_OUT.SEND_PUBLSIH:
			PublishSendList[PublishSendListCount] := i;
			PublishSendListCount := PublishSendListCount + 1;
			
		STEPS_OUT.WAIT_PUBACK:
			IF OutData[i].TimeOutStarted AND OutData[i].TimeOut.Q THEN
				PushError(newError:= ERRORS.REPEAT_PUBLISH_PUBACK, text:= CONCAT(STR1 := CONCAT(STR1:= 'Slot:', STR2:= TO_STRING(i)),
							 STR2:= CONCAT(STR1:=', PAKET:', STR2:=TO_STRING(OutData[i].InDataFromFb^.PaketId ))));
				//timeout, need repead
				OutData[i].InDataFromFb^.DUP := TRUE;
				OutData[i].step := STEPS_OUT.SEND_PUBLSIH;//repeat publish
				RepeatedPublish := RepeatedPublish + 1;
				OutData[i].TimeOutStarted := FALSE;
			END_IF
			
		STEPS_OUT.WAIT_PUBREC:
			IF OutData[i].TimeOutStarted AND OutData[i].TimeOut.Q THEN
				PushError(newError:= ERRORS.REPEAT_PUBLISH_PUBREC, text:= CONCAT(STR1 := CONCAT(STR1:= 'Slot:', STR2:= TO_STRING(i)),
							 STR2:= CONCAT(STR1:=', PAKET:', STR2:=TO_STRING(OutData[i].InDataFromFb^.PaketId ))));
				//timeout, need repead
				OutData[i].InDataFromFb^.DUP := TRUE;
				OutData[i].step := STEPS_OUT.SEND_PUBLSIH;//repeat publish
				RepeatedPublish := RepeatedPublish + 1;
				OutData[i].TimeOutStarted := FALSE;
			END_IF
			
		STEPS_OUT.SEND_PUBREL:
			PubrelSendList[PubrelSendListCount] := i;
			PubrelSendListCount := PubrelSendListCount + 1;
			
		STEPS_OUT.WAIT_PUBCOMP:
			IF OutData[i].TimeOutStarted AND OutData[i].TimeOut.Q THEN
				//timeout, need repead
				OutData[i].step := STEPS_OUT.SEND_PUBREL;//repeat pubrel
				RepeatedPubrel := RepeatedPubrel + 1;
				OutData[i].TimeOutStarted := FALSE;
				OutData[i].PUBRELRepeatCounter := OutData[i].PUBRELRepeatCounter + 1;
				IF OutData[i].PUBRELRepeatCounter >= MyConstants.MAX_PUBREL_REPEATS THEN
					OutData[i].PUBRELRepeatCounter := 0;
					//resend publish
					OutData[i].step := STEPS_OUT.SEND_PUBLSIH;
					OutData[i].InDataFromFb^.DUP := TRUE;
					RepeatedPublishsAfterPubrel := RepeatedPublishsAfterPubrel + 1;
					PushError(newError:= ERRORS.REPEAT_PUBLISH_PUBCOMP, text:= CONCAT(STR1 := CONCAT(STR1:= 'Slot:', STR2:= TO_STRING(i)),
							 STR2:= CONCAT(STR1:=', PAKET:', STR2:=TO_STRING(OutData[i].InDataFromFb^.PaketId ))));
				ELSE
					PushError(newError:= ERRORS.REPEAT_PUBREL, text:= CONCAT(STR1 := CONCAT(STR1:= 'Slot:', STR2:= TO_STRING(i)),
							 STR2:= CONCAT(STR1:=', PAKET:', STR2:=TO_STRING(OutData[i].InDataFromFb^.PaketId ))));
				END_IF
			END_IF
		IF NOT (OutData[i].step = STEPS_OUT.WAIT_DATA) THEN
			TempSlotsWorking := TempSlotsWorking + 1;
		END_IF
	END_CASE
	//make sure timer is set to 0 if timeout resetet
	OutData[i].TimeOut(IN:= OutData[i].TimeOutStarted, PT:= MyConstants.REPEAT_TIMEOUT);
END_FOR

//now sort the arrays...
IF PublishSendListCount > 1 THEN
	FOR i := 0 TO PublishSendListCount - 1 DO
		tmpLowest := 16#FFFF;
		minIndex := i;
		FOR j := i TO PublishSendListCount - 1 DO
			IF OutData[PublishSendList[j]].PUBLISHOrder < tmpLowest THEN
				minIndex := j;
				tmpLowest := OutData[PublishSendList[j]].PUBLISHOrder;
			END_IF
		END_FOR
		IF minIndex <> i THEN
			//hier tauschen
			j := PublishSendList[minIndex];
			PublishSendList[minIndex] := PublishSendList[i];
			PublishSendList[i] := j;
		END_IF
	END_FOR
END_IF

IF PubrelSendListCount > 1 THEN
	FOR i := 0 TO PubrelSendListCount - 1 DO
		tmpLowest := 16#FFFF;
		minIndex := i;
		FOR j := i TO PubrelSendListCount - 1 DO
			IF OutData[PubrelSendList[j]].PUBRECOrder < tmpLowest THEN
				minIndex := j;
				tmpLowest := OutData[PubrelSendList[j]].PUBRECOrder;
			END_IF
		END_FOR
		IF minIndex <> i THEN
			//hier tauschen
			j := PubrelSendList[minIndex];
			PubrelSendList[minIndex] := PubrelSendList[i];
			PubrelSendList[i] := j;
		END_IF
	END_FOR
END_IF

//Hamdel PubrelOrderIndexCounter
IF PubrelOrderIndexCounter > MyConstants.REORDER_VALUE THEN 
	PushError(newError:= ERRORS.REORDER_PUBREC , text:= '');
	//do it brute force, just sub 20000 to every value...
	FOR i := 0 TO MyConstants.QoS_BUFFER_SIZE - 1 DO
		OutData[i].PUBRECOrder := OutData[i].PUBRECOrder - MyConstants.SUBSTRACTION_VALUE;
	END_FOR
	PubrelOrderIndexCounter := MyConstants.REORDER_VALUE - MyConstants.SUBSTRACTION_VALUE + 1;
END_IF
//Hamdel PublishOrderIndexCounter
IF OutgoingPublishOrderIndexCounter > MyConstants.REORDER_VALUE THEN 
	PushError(newError:= ERRORS.REORDER_PUBLISH_OUTGOING, text:= '');
	//do it brute force, just sub 20000 to every value...
	FOR i := 0 TO MyConstants.QoS_BUFFER_SIZE - 1 DO
		OutData[i].PUBLISHOrder := OutData[i].PUBLISHOrder - MyConstants.SUBSTRACTION_VALUE;
	END_FOR
	OutgoingPublishOrderIndexCounter := MyConstants.REORDER_VALUE - MyConstants.SUBSTRACTION_VALUE + 1;
END_IF

OutSlotsWorking := TempSlotsWorking;
                
END_METHOD

METHOD StateMashineIn
  VAR_INPUT
    MQTT_IN_OUT : POINTER TO MQTT_IN_OUT;
  END_VAR
  VAR
    i : UINT;
    j : UINT;
    TempSlotsWorking : UINT;
    tmpLowest : UINT;
    minIndex : UINT;
  END_VAR
                  
GVL_MQTT.ProgNum := PROG_NUM.STATE_MASHINE_IN;
//Handle State Mashines
PubackSendListCount := 0;
PubrecSendListCount := 0;
PubcompSendListCount := 0;
TempSlotsWorking := 0;
FOR i := 0 TO MyConstants.QoS_BUFFER_SIZE - 1 DO
	//do Timers...
	InData[i].TimeOut(IN:= InData[i].TimeOutStarted, PT:= MyConstants.REPEAT_TIMEOUT);
	IF NOT (InData[i].step = STEPS_IN.WAIT_DATA) THEN
		TempSlotsWorking := TempSlotsWorking + 1;
	END_IF  
	CASE InData[i].step OF
		STEPS_IN.WAIT_DATA:;
		STEPS_IN.WAIT_PUBREL:
		IF InData[i].TimeOut.Q THEN
			InData[i].step := STEPS_IN.SEND_PUBREC;
			InData[i].TimeOutStarted := FALSE;
			CountRepeatetPubrec := CountRepeatetPubrec + 1;
			PUBREC_ERROR_ID_BUFFER[PUBREC_ERROR_INDEX] := InData[i].PaketID; 
			PUBREC_ERROR_INDEX := PUBREC_ERROR_INDEX + 1;
			InData[i].CountPubrecRepeat := InData[i].CountPubrecRepeat + 1;
				
			IF InData[i].CountPubrecRepeat > COUNT_MAX_PUBREC_REPEAT_TO_DISCHARGE THEN
				InData[i].CountPubrecRepeat := 0;
				InData[i].step := STEPS_IN.WAIT_DATA;
				PushError(newError:= ERRORS.PUBEC_DISCHARGE, text:= CONCAT(STR1 := CONCAT(STR1:= 'Slot:', STR2:= TO_STRING(i)),
							 STR2:= CONCAT(STR1:=', PAKET:', STR2:=TO_STRING(InData[i].PaketID))));
			
			ELSE
				PushError(newError:= ERRORS.REORDER_PUBREC, text:= CONCAT(STR1 := CONCAT(STR1:= 'Slot:', STR2:= TO_STRING(i)),
							 STR2:= CONCAT(STR1:=', PAKET:', STR2:=TO_STRING(InData[i].PaketID))));
			
			END_IF
			IF PUBREC_ERROR_INDEX >= PUBREC_ERROR_ID_BUFFER_SIZE THEN
				PUBREC_ERROR_INDEX := 0;
			END_IF
		END_IF
		STEPS_IN.SEND_PUBACK:
			PubackSendList[PubackSendListCount] := i;
			PubackSendListCount := PubackSendListCount + 1;
			
		STEPS_IN.SEND_PUBREC:
			PubrecSendList[PubrecSendListCount] := i;
			PubrecSendListCount := PubrecSendListCount + 1;
		
		STEPS_IN.SEND_PUBCOMP:
			PubcompSendList[PubcompSendListCount] := i;
			PubcompSendListCount := PubcompSendListCount + 1;
		
	END_CASE
	//make sure timer is set to 0 if timeout resetet
	InData[i].TimeOut(IN:= InData[i].TimeOutStarted, PT:= MyConstants.REPEAT_TIMEOUT);
END_FOR


//now sort the arrays...
IF PubackSendListCount > 1 THEN
	FOR i := 0 TO PubackSendListCount - 1 DO
		tmpLowest := 16#FFFF;
		minIndex := i;
		FOR j := i TO PubackSendListCount - 1 DO
			IF InData[PubackSendList[j]].PUBLISHOrder < tmpLowest THEN
				minIndex := j;
				tmpLowest := InData[PubackSendList[j]].PUBLISHOrder;
			END_IF
		END_FOR
		IF minIndex <> i THEN
			//hier tauschen
			j := PubackSendList[minIndex];
			PubackSendList[minIndex] := PubackSendList[i];
			PubackSendList[i] := j;
		END_IF
	END_FOR
END_IF

IF PubrecSendListCount > 1 THEN
	FOR i := 0 TO PubrecSendListCount - 1 DO
		tmpLowest := 16#FFFF;
		minIndex := i;
		FOR j := i TO PubrecSendListCount - 1 DO
			IF InData[PubrecSendList[j]].PUBLISHOrder < tmpLowest THEN
				minIndex := j;
				tmpLowest := InData[PubrecSendList[j]].PUBLISHOrder;
			END_IF
		END_FOR
		IF minIndex <> i THEN
			//hier tauschen
			j := PubrecSendList[minIndex];
			PubrecSendList[minIndex] := PubrecSendList[i];
			PubrecSendList[i] := j;
		END_IF
	END_FOR
END_IF


IF PubcompSendListCount > 1 THEN
	FOR i := 0 TO PubcompSendListCount - 1 DO
		tmpLowest := 16#FFFF;
		minIndex := i;
		FOR j := i TO PubcompSendListCount - 1 DO
			IF InData[PubcompSendList[j]].PUBCOMPOrder < tmpLowest THEN
				minIndex := j;
				tmpLowest := InData[PubcompSendList[j]].PUBCOMPOrder;
			END_IF
		END_FOR
		IF minIndex <> i THEN
			//hier tauschen
			j := PubcompSendList[minIndex];
			PubcompSendList[minIndex] := PubcompSendList[i];
			PubcompSendList[i] := j;
		END_IF
	END_FOR
END_IF
//Hamdel PublishOrderIndexCounter
IF IncomingPublishOrderIndexCounter > MyConstants.REORDER_VALUE THEN 
	PushError(newError:= ERRORS.REODER_PUBLISH_INCOMMING , text:= '');
			
	//do it brute force, just sub 20000 to every value...
	FOR i := 0 TO MyConstants.QoS_BUFFER_SIZE - 1 DO
		InData[i].PUBLISHOrder := InData[i].PUBLISHOrder - MyConstants.SUBSTRACTION_VALUE;
	END_FOR
	IncomingPublishOrderIndexCounter := MyConstants.REORDER_VALUE - MyConstants.SUBSTRACTION_VALUE + 1;
END_IF

//Hamdel PublishOrderIndexCounter
IF PubcompOrderIndexCounter > MyConstants.REORDER_VALUE THEN 
	PushError(newError:= ERRORS.REORDER_PUBCOMP, text:= '');
	
	//do it brute force, just sub 20000 to every value...
	FOR i := 0 TO MyConstants.QoS_BUFFER_SIZE - 1 DO
		InData[i].PUBCOMPOrder := InData[i].PUBCOMPOrder - MyConstants.SUBSTRACTION_VALUE;
	END_FOR
	PubcompOrderIndexCounter := MyConstants.REORDER_VALUE - MyConstants.SUBSTRACTION_VALUE + 1;
END_IF

InSlotsWorking := TempSlotsWorking;
                
END_METHOD

METHOD BuildPublishPaket : BOOL
  VAR_INPUT
    PaketData : POINTER TO PAKET_DATA;
  END_VAR
  VAR
    idx : UINT;
  END_VAR
                  (*now change to realy big topics and payloads, do that to big topics and payloads transmitted splitted*)

BuildPublishPaket := FALSE;
IF StepBuildPublish = 0 THEN
	StepBuildPublish := 10; 
END_IF

idx := COM.S_BUF.SIZE;
//check if buffer is big enought for control, remainig length, topic size....
IF StepBuildPublish = 10 THEN

	IF (6 + COM.S_BUF.SIZE)
		 > TRANSMIT_BUFFER_SIZE THEN//only check if header fits into buffer...
		 CountCantSendPublishBufferToFull := CountCantSendPublishBufferToFull + 1;
		RETURN;	
	END_IF
	COM.S_BUF.BUFFER[idx] := MESSAGETYPE.PUBLISH;//set type
	IF PaketData^.DUP THEN//insert DUP bit
		COM.S_BUF.BUFFER[idx] := COM.S_BUF.BUFFER[idx] OR 2#1000;
	END_IF 
	COM.S_BUF.BUFFER[idx] := COM.S_BUF.BUFFER[idx] OR SHL(PaketData^.MessageQoS,1);
	IF PaketData^.MessageRetain THEN
		COM.S_BUF.BUFFER[idx] := COM.S_BUF.BUFFER[idx] OR 2#1;
	END_IF
	//do remainig lenght... 

	idx := idx + 2 + DoRemainingLengthBevor(buffer:= ADR(COM.S_BUF.BUFFER[idx]), SizeTopic:= PaketData^.MqttTopicLength, SizePayload:= PaketData^.MqttPayloadLength, InQoS:= PaketData^.MessageQoS);

	StepBuildPublish := 20;
END_IF

IF StepBuildPublish = 20 THEN
	GVL_MQTT.ProgNum := PROG_NUM.SendOutDataInsertTopic;
	//insert topic
	InsertSplitTopic(
		topic:= PaketData^.MqttTopic, 
		len:= PaketData^.MqttTopicLength, 
		buff:= ADR(COM.S_BUF.BUFFER), 
		pos:= idx, 
		size:= NETWORK_BUFFER_LONG_SIZE);
	CASE InsertSplitTopic.state OF
		INSERT_SPLIT_RETURN.INSERT_DONE:
			StepBuildPublish := 30;
		INSERT_SPLIT_RETURN.INSERT_ERROR:
			StepBuildPublish := 0;
			InsertSplitTopic.reset();
			RETURN;
		INSERT_SPLIT_RETURN.INSERT_PENDING:
			//here do nothing, just wait
		ELSE
			InsertSplitTopic.reset();
			StepBuildPublish := 0;
			RETURN;
	END_CASE
	idx := InsertSplitTopic.new_pos;
END_IF
IF StepBuildPublish = 30 THEN
	IF PaketData^.MessageQoS > 0 THEN//QoS is more then 0
		IF (2 + idx)//insert paket identifier
		 < TRANSMIT_BUFFER_SIZE THEN//enough space for identifier?
			COM.S_BUF.BUFFER[idx] := OSCAT_BASIC.BYTE_OF_DWORD(in:= PaketData^.PaketId, N:= 1);
			idx := idx + 1;
			COM.S_BUF.BUFFER[idx] := OSCAT_BASIC.BYTE_OF_DWORD(in:= PaketData^.PaketId, N:= 0);
			idx := idx + 1;
			StepBuildPublish := 40;
		END_IF
	ELSE
		StepBuildPublish := 40;
	END_IF
END_IF

IF StepBuildPublish = 40 THEN
	GVL_MQTT.ProgNum := PROG_NUM.SendOutDataInsertPayload;
	//now insert payload
	IF PaketData^.MqttPayloadLength > 0 THEN
		//insert payload
		InsertSplitPayload(
			payload:= PaketData^.MqttPayload, 
			len:= PaketData^.MqttPayloadLength, 
			buff:= ADR(COM.S_BUF.BUFFER), 
			pos:= idx, 
			size:= NETWORK_BUFFER_LONG_SIZE);
		CASE InsertSplitPayload.state OF
			INSERT_SPLIT_RETURN.INSERT_DONE:
				StepBuildPublish := 0;
				BuildPublishPaket := TRUE;
			INSERT_SPLIT_RETURN.INSERT_ERROR:
				StepBuildPublish := 0;
				InsertSplitPayload.reset();
				RETURN;
			INSERT_SPLIT_RETURN.INSERT_PENDING:
				//here do nothing, just wait
				//or handle timeout....
			ELSE
				InsertSplitPayload.reset();
				StepBuildPublish := 0;
				RETURN;
		END_CASE
		idx := InsertSplitPayload.new_pos;
	ELSE
		StepBuildPublish := 0;
		BuildPublishPaket := TRUE;
	END_IF
END_IF
COM.S_BUF.SIZE := idx;

                
END_METHOD

METHOD MoveBufferForSplitPaket
  VAR_INPUT
    idx : UINT;
  END_VAR
  VAR
    BytesToMove : UINT;
  END_VAR
                  GVL_MQTT.ProgNum := PROG_NUM.MoveBuffer;
BytesToMove := COM.R_BUF.SIZE - idx;
CountBufferMoves := CountBufferMoves + 1;
MEM.MemMove(pSource:= ADR(com.R_BUF.BUFFER[idx]), pDestination:= ADR(com.R_BUF.BUFFER), uiNumberOfBytes:= BytesToMove);
COM.R_BUF.SIZE := BytesToMove;//manipulate size....

                
END_METHOD

METHOD BuildSubscribePaket : BOOL
  VAR_INPUT
    PaketData : POINTER TO PAKET_DATA;
  END_VAR
  VAR
    idx : UINT;
  END_VAR
                  BuildSubscribePaket := FALSE;
IF  StepBuildSubscribe = 0 THEN
	StepBuildSubscribe := 10;
END_IF

idx := COM.S_BUF.SIZE;
IF StepBuildSubscribe = 10 THEN
	IF (6 + COM.S_BUF.SIZE)
	 > TRANSMIT_BUFFER_SIZE THEN//only check if header fits into buffer...
		 RETURN;
	END_IF
	idx := COM.S_BUF.SIZE;
	COM.S_BUF.BUFFER[idx] := MESSAGETYPE.SUBSCRIBE OR 2#10;//set type, for 2#10 see subscribe doku
	idx := idx + 2 + DoRemainingLengthBevor(buffer:= ADR(COM.S_BUF.BUFFER[idx]), SizeTopic:= PaketData^.MqttTopicLength, SizePayload:= 1, InQoS:= QoS.AtLeastOnce);
	COM.S_BUF.BUFFER[idx] := OSCAT_BASIC.BYTE_OF_DWORD(in:= PaketData^.PaketId, N:= 1);
	idx := idx + 1;
	COM.S_BUF.BUFFER[idx] := OSCAT_BASIC.BYTE_OF_DWORD(in:= PaketData^.PaketId, N:= 0);
	idx := idx + 1;
	StepBuildSubscribe := 20;
END_IF


IF StepBuildSubscribe = 20 THEN
	//insert topic
	InsertSplitTopic(
		topic:= PaketData^.MqttTopic, 
		len:= PaketData^.MqttTopicLength, 
		buff:= ADR(COM.S_BUF.BUFFER), 
		pos:= idx, 
		size:= NETWORK_BUFFER_LONG_SIZE);
	CASE InsertSplitTopic.state OF
		INSERT_SPLIT_RETURN.INSERT_DONE:
			StepBuildSubscribe := 30;
		INSERT_SPLIT_RETURN.INSERT_ERROR:
			StepBuildSubscribe := 0;
			InsertSplitTopic.reset();
			RETURN;
		INSERT_SPLIT_RETURN.INSERT_PENDING:
			//here do nothing, just wait
		ELSE
			InsertSplitTopic.reset();
			StepBuildSubscribe := 0;
			RETURN;
	END_CASE
	idx := InsertSplitTopic.new_pos;
END_IF

IF StepBuildSubscribe = 30 THEN

	IF (1 + idx)
	 > TRANSMIT_BUFFER_SIZE THEN//only check if qos fits into buffer...
		 RETURN;
	 END_IF
	//insert QoS
	COM.S_BUF.BUFFER[idx] := PaketData^.MessageQoS;
	idx := idx + 1;
	StepBuildSubscribe := 0;
	BuildSubscribePaket := TRUE;
END_IF

COM.S_BUF.SIZE := idx;
                
END_METHOD

METHOD BuildUnsubscribePaket : BOOL
  VAR_INPUT
    PaketData : POINTER TO PAKET_DATA;
  END_VAR
  VAR
    idx : UINT;
  END_VAR
                  BuildUnsubscribePaket := FALSE;

IF  StepBuildUnsubscribe = 0 THEN
	StepBuildUnsubscribe := 10;
END_IF

idx := COM.S_BUF.SIZE;
IF StepBuildUnsubscribe = 10 THEN
	IF (6 + COM.S_BUF.SIZE)
	 > TRANSMIT_BUFFER_SIZE THEN//only check if header fits into buffer...
		 RETURN;
	END_IF
	idx := COM.S_BUF.SIZE;
	COM.S_BUF.BUFFER[idx] := MESSAGETYPE.UNSUBSCRIBE OR 2#10;//set type, for 2#10 see subscribe doku
	idx := idx + 2 + DoRemainingLengthBevor(buffer:= ADR(COM.S_BUF.BUFFER[idx]), SizeTopic:= PaketData^.MqttTopicLength, SizePayload:= 0, InQoS:= QoS.AtLeastOnce);
	COM.S_BUF.BUFFER[idx] := OSCAT_BASIC.BYTE_OF_DWORD(in:= PaketData^.PaketId, N:= 1);
	idx := idx + 1;
	COM.S_BUF.BUFFER[idx] := OSCAT_BASIC.BYTE_OF_DWORD(in:= PaketData^.PaketId, N:= 0);
	idx := idx + 1;
	StepBuildUnsubscribe := 20;
END_IF


IF StepBuildUnsubscribe = 20 THEN
	//insert topic
	InsertSplitTopic(
		topic:= PaketData^.MqttTopic, 
		len:= PaketData^.MqttTopicLength, 
		buff:= ADR(COM.S_BUF.BUFFER), 
		pos:= idx, 
		size:= NETWORK_BUFFER_LONG_SIZE);
	CASE InsertSplitTopic.state OF
		INSERT_SPLIT_RETURN.INSERT_DONE:
			StepBuildUnsubscribe := 0;
			BuildUnsubscribePaket := TRUE;
		INSERT_SPLIT_RETURN.INSERT_ERROR:
			StepBuildUnsubscribe := 0;
			InsertSplitTopic.reset();
			RETURN;
		INSERT_SPLIT_RETURN.INSERT_PENDING:
			//here do nothing, just wait
		ELSE
			InsertSplitTopic.reset();
			StepBuildUnsubscribe := 0;
			RETURN;
	END_CASE
	idx := InsertSplitTopic.new_pos;
END_IF

COM.S_BUF.SIZE := idx;

                
END_METHOD

METHOD SendOutData
  VAR_INPUT
    MQTT_IN_OUT : POINTER TO MQTT_IN_OUT;  (* StepData:POINTER TO MQTT_OUT_DATA; *)
  END_VAR
  VAR
    SomethingIsBlocking : BOOL;
    i : UINT;
  END_VAR
                  IF NOT SendFree THEN RETURN; END_IF
GVL_MQTT.ProgNum := PROG_NUM.SendOutData;

SomethingIsBlocking := SendInfos.PublishBlocking OR SendInfos.SubscribeBlocking OR SendInfos.UnsubscribeBlocking;

//Prio for Timeout Paket
IF  NOT (COM.S_BUF.SIZE + SIZE_PINGREQ > TRANSMIT_BUFFER_SIZE) AND SendInfos.PingNeeded AND NOT SomethingIsBlocking THEN
	SendInfos.PingNeeded := FALSE;
	COM.S_BUF.BUFFER[COM.S_BUF.SIZE] := MESSAGETYPE.PINGREQ;
	COM.S_BUF.BUFFER[COM.S_BUF.SIZE + 1] := 0;//no more length 	
	COM.S_BUF.SIZE := COM.S_BUF.SIZE + SIZE_PINGREQ;//small ping paket
	OutData[SendInfos.PingIndex].TimeOutStarted := TRUE;//start Timeout
END_IF
IF NOT COM.S_BUF.SIZE = 0 THEN 
	CountOutSendNotFree := CountOutSendNotFree + 1;
END_IF
//next Prio send Pubrel 
IF PubrelSendListCount > 0 AND NOT SomethingIsBlocking THEN
	FOR i := 0 TO PubrelSendListCount - 1 DO
		IF NOT (COM.S_BUF.SIZE + SIZE_PUBREL > TRANSMIT_BUFFER_SIZE) THEN
			COM.S_BUF.BUFFER[COM.S_BUF.SIZE] := MESSAGETYPE.PUBREL OR 2#10;//set type and Reserved bits
			COM.S_BUF.BUFFER[COM.S_BUF.SIZE + 1] := 2;
			COM.S_BUF.BUFFER[COM.S_BUF.SIZE + 2] := OSCAT_BASIC.BYTE_OF_DWORD(in:= OutData[PubrelSendList[i]].InDataFromFb^.PaketId, N:= 1);
			COM.S_BUF.BUFFER[COM.S_BUF.SIZE + 3] := OSCAT_BASIC.BYTE_OF_DWORD(in:= OutData[PubrelSendList[i]].InDataFromFb^.PaketId, N:= 0);
			COM.S_BUF.SIZE := COM.S_BUF.SIZE + SIZE_PUBREL;
			OutData[PubrelSendList[i]].step := STEPS_OUT.WAIT_PUBCOMP;
			OutData[PubrelSendList[i]].TimeOutStarted := TRUE;//start Timeout			
		ELSE
			EXIT;
		END_IF 
	END_FOR
END_IF

//send Unsubscribe
IF SendInfos.UnsubscribeNeeded AND (NOT SomethingIsBlocking OR SendInfos.UnsubscribeBlocking) THEN
	IF NOT BuildUnsubscribePaket(PaketData:= OutData[SendInfos.UnsubscribeIndex].InDataFromFb) THEN
		SendInfos.UnsubscribeBlocking := TRUE;
	ELSE
		SendInfos.UnsubscribeBlocking := FALSE;
		SendInfos.UnsubscribeNeeded := FALSE;
		OutData[SendInfos.UnsubscribeIndex].TimeOutStarted := TRUE;
		OutData[SendInfos.UnsubscribeIndex].step := STEPS_OUT.WAIT_UNSUBACK;
	END_IF
END_IF

//send Subscribe
IF SendInfos.SubscribeNeeded AND (NOT SomethingIsBlocking OR SendInfos.SubscribeBlocking) THEN
	IF NOT BuildSubscribePaket(PaketData:= OutData[SendInfos.SubscribeIndex].InDataFromFb) THEN
		SendInfos.SubscribeBlocking := TRUE;
	ELSE
		SendInfos.SubscribeBlocking := FALSE;
		SendInfos.SubscribeNeeded := FALSE;
		OutData[SendInfos.SubscribeIndex].TimeOutStarted := TRUE;
		OutData[SendInfos.SubscribeIndex].step := STEPS_OUT.WAIT_SUBACK;
	END_IF
END_IF
//send pending Publish 
IF SendInfos.PublishBlocking THEN
	IF BuildPublishPaket(PaketData:= OutData[SendInfos.PublishBlockingIndex].InDataFromFb) THEN
		SendInfos.PublishBlocking := FALSE;
		PublishSendDone(slot:=ADR(OutData[SendInfos.PublishBlockingIndex]));
	END_IF
END_IF

IF (PublishSendListCount > 0 AND NOT SomethingIsBlocking) THEN
	//handle pendig publisah packet
	//handle new publish packet
	FOR i := 0 TO PublishSendListCount - 1 DO
		IF NOT BuildPublishPaket(PaketData:= OutData[PublishSendList[i]].InDataFromFb) THEN
			SendInfos.PublishBlocking := TRUE;
			SendInfos.PublishBlockingIndex := PublishSendList[i];
			EXIT;
		ELSE 
			SendInfos.PublishBlocking := FALSE;
			PublishSendDone(slot:=ADR(OutData[PublishSendList[i]]));
		END_IF
	END_FOR
END_IF
                
END_METHOD

METHOD SendInData
  VAR_INPUT
    MQTT_IN_OUT : POINTER TO MQTT_IN_OUT;
  END_VAR
  VAR
    i : UINT;
  END_VAR
                  IF NOT SendFree THEN RETURN; END_IF

GVL_MQTT.ProgNum := PROG_NUM.SendInData;

IF NOT COM.S_BUF.SIZE = 0 THEN 
	CountInSendNotFree := CountInSendNotFree + 1;
END_IF

IF PubackSendListCount > 0 THEN
	FOR i := 0 TO PubackSendListCount - 1 DO
		IF NOT (COM.S_BUF.SIZE + SIZE_PUBACK > TRANSMIT_BUFFER_SIZE)  THEN
			COM.S_BUF.BUFFER[COM.S_BUF.SIZE] := MESSAGETYPE.PUBACK;
			COM.S_BUF.BUFFER[COM.S_BUF.SIZE + 1] := 2;//length of 2
			COM.S_BUF.BUFFER[COM.S_BUF.SIZE + 2] := OSCAT_BASIC.BYTE_OF_DWORD(in:= InData[PubackSendList[i]].PaketID, N:= 1);
			COM.S_BUF.BUFFER[COM.S_BUF.SIZE + 3] := OSCAT_BASIC.BYTE_OF_DWORD(in:= InData[PubackSendList[i]].PaketID, N:= 0);
			COM.S_BUF.SIZE := COM.S_BUF.SIZE + SIZE_PUBACK;//Paket size allways 4!
			InData[PubackSendList[i]].step := STEPS_IN.WAIT_DATA;
			MqttsDoneIo := MqttsDoneIo + 1;	
		ELSE
			EXIT;
		END_IF
	END_FOR
	
END_IF

IF PubcompSendListCount > 0 THEN
	FOR i := 0 TO PubcompSendListCount - 1 DO
		IF NOT (COM.S_BUF.SIZE + SIZE_PUBCOMP > TRANSMIT_BUFFER_SIZE) THEN	
			COM.S_BUF.BUFFER[COM.S_BUF.SIZE] := MESSAGETYPE.PUBCOMP;
			COM.S_BUF.BUFFER[COM.S_BUF.SIZE + 1] := 2;//length of 2
			COM.S_BUF.BUFFER[COM.S_BUF.SIZE + 2] := OSCAT_BASIC.BYTE_OF_DWORD(in:= InData[PubcompSendList[i]].PaketID, N:= 1);
			COM.S_BUF.BUFFER[COM.S_BUF.SIZE + 3] := OSCAT_BASIC.BYTE_OF_DWORD(in:= InData[PubcompSendList[i]].PaketID, N:= 0);
			COM.S_BUF.SIZE := COM.S_BUF.SIZE + SIZE_PUBCOMP;//Paket size allways 4!
			InData[PubcompSendList[i]].step := STEPS_IN.WAIT_DATA;
			MqttsDoneIo := MqttsDoneIo + 1;
		ELSE
			EXIT;
		END_IF
	END_FOR
END_IF

IF PubrecSendListCount > 0 THEN
	FOR i := 0 TO PubrecSendListCount - 1 DO
		IF NOT (COM.S_BUF.SIZE + SIZE_PUBREC > TRANSMIT_BUFFER_SIZE) THEN
			COM.S_BUF.BUFFER[COM.S_BUF.SIZE] := MESSAGETYPE.PUBREC;
			COM.S_BUF.BUFFER[COM.S_BUF.SIZE + 1] := 2;//length of 2
			COM.S_BUF.BUFFER[COM.S_BUF.SIZE + 2] := OSCAT_BASIC.BYTE_OF_DWORD(in:= InData[PubrecSendList[i]].PaketID, N:= 1);
			COM.S_BUF.BUFFER[COM.S_BUF.SIZE + 3] := OSCAT_BASIC.BYTE_OF_DWORD(in:= InData[PubrecSendList[i]].PaketID, N:= 0);
			COM.S_BUF.SIZE := COM.S_BUF.SIZE + SIZE_PUBREC;//Paket size allways 4!
			InData[PubrecSendList[i]].step := STEPS_IN.WAIT_PUBREL;
			InData[PubrecSendList[i]].TimeOutStarted := TRUE;
		ELSE
			EXIT;
		END_IF
	END_FOR
END_IF

                
END_METHOD

METHOD ParseIncoming
  VAR_INPUT
    MQTT_IN_OUT : POINTER TO MQTT_IN_OUT;
  END_VAR
  VAR
    I : UINT;
    j : UINT;
    idx : UINT := 0;
    ReceivePakteType : MESSAGETYPE;  (* idxFromParsePublish:UINT := 0; *)
    ReceivePaketID : WORD;
    BufferMoveDone : BOOL;
    PaketFound : BOOL;
  END_VAR
                  GVL_MQTT.ProgNum := PROG_NUM.ParseIncomming;
IF COM.R_BUF.SIZE > 0 THEN
	REPEAT
		
		PaketFound := FALSE;
		HelperLastPaktetForUnkownPaket := ReceivePakteType;
		ReceivePakteType := COM.R_BUF.BUFFER[idx] AND 16#F0;
		 
		CASE ReceivePakteType OF
			MESSAGETYPE.PUBLISH:
			//new way, move every publish to receive buffer, and then pars it.
			//outgoing payload pointer is then set to start of payload in the buffer....
				BufferMoveDone := CheckLenghtBuffer(IdxIn:= idx);
				IF NOT BufferMoveDone THEN
					
					idx := ParseIncomingPublish(MQTT_IN_OUT:= MQTT_IN_OUT, idx:= idx,
											BufferIn:= ADR(COM.R_BUF.BUFFER), BufferSize:= COM.R_BUF.SIZE,
											NetworkBuffer:= TRUE);

				END_IF
			MESSAGETYPE.PUBREL:
				BufferMoveDone := CheckLenghtBuffer(IdxIn:= idx);
				IF NOT BufferMoveDone THEN
					//get Paket ID
					ReceivePaketID := DWORD_TO_WORD(OSCAT_BASIC.DWORD_OF_BYTE(B3:= 0, B2:= 0, 
						B1:= COM.R_BUF.BUFFER[idx + 2],
						B0:= COM.R_BUF.BUFFER[idx + 3]));
					//find Paket
					FOR i := 0 TO MyConstants.QoS_BUFFER_SIZE - 1 DO
						IF InData[i].PaketID = ReceivePaketID THEN
							InData[i].step := STEPS_IN.SEND_PUBCOMP;
							InData[i].TimeOutStarted := FALSE;
							PubcompOrderIndexCounter := PubcompOrderIndexCounter;
							InData[i].PUBCOMPOrder := PubcompOrderIndexCounter;
							PaketFound := TRUE;
							EXIT;
						END_IF
						//
					END_FOR
					IF NOT PaketFound THEN
						CountReceivePubrelUnknown := CountReceivePubrelUnknown + 1;
					END_IF
					idx := idx + SIZE_PUBREL;
				END_IF
			MESSAGETYPE.PINGRESP:
				ResetPingTime();
				PingRequestet := FALSE;
				OutData[PingSlot].step := STEPS_OUT.WAIT_DATA;//can get new data
				OutData[PingSlot].TimeOutStarted := FALSE;
				idx := idx + SIZE_PINGRESP;
			MESSAGETYPE.UNSUBACK:
				BufferMoveDone := CheckLenghtBuffer(IdxIn:= idx);
				IF NOT BufferMoveDone THEN
					//get Paket ID
					ReceivePaketID := DWORD_TO_WORD(OSCAT_BASIC.DWORD_OF_BYTE(B3:= 0, B2:= 0, 
						B1:= COM.R_BUF.BUFFER[idx + 2],
						B0:= COM.R_BUF.BUFFER[idx + 3]));
					//find Paket
					FOR i := 0 TO MyConstants.QoS_BUFFER_SIZE - 1 DO
						IF OutData[i].step = STEPS_OUT.WAIT_UNSUBACK THEN //make sure pointer is vailid
							IF OutData[i].InDataFromFb^.PaketId = ReceivePaketID THEN
								OutData[i].InDataFromFb^.SendSucsess := TRUE;
								OutData[i].step := STEPS_OUT.WAIT_DATA;//can get new data
								OutData[i].TimeOutStarted := FALSE;
								MqttsDoneIo := MqttsDoneIo + 1;
								PaketFound := TRUE;
								//now kick of Callback
								FOR j := 0 TO CALLBACKS_BUFFER_SIZE - 1 DO
									IF SubscribeCallbacks[j].Callback = OutData[i].InDataFromFb^.Callback  THEN
										//callback found, now kill it...
										SubscribeCallbacks[j].free := TRUE;
										SubscribeCallbacks[j].Callback := 0;
										EXIT;
									END_IF
								END_FOR
								EXIT;
							END_IF
						END_IF
						//
					END_FOR
					IF NOT PaketFound THEN
						CountReceiveUnsubackUnknown := CountReceiveUnsubackUnknown + 1;
					END_IF
					idx := idx + SIZE_UNSUBACK;	
				END_IF
				
			MESSAGETYPE.SUBACK:
				BufferMoveDone := CheckLenghtBuffer(IdxIn:= idx);
				IF NOT BufferMoveDone THEN
					//get Paket ID
					ReceivePaketID := DWORD_TO_WORD(OSCAT_BASIC.DWORD_OF_BYTE(B3:= 0, B2:= 0, 
						B1:= COM.R_BUF.BUFFER[idx + 2],
						B0:= COM.R_BUF.BUFFER[idx + 3]));
					//find Paket
					FOR i := 0 TO MyConstants.QoS_BUFFER_SIZE - 1 DO
						IF OutData[i].step = STEPS_OUT.WAIT_SUBACK THEN //make sure pointer is vailid
							IF OutData[i].InDataFromFb^.PaketId = ReceivePaketID THEN
								OutData[i].InDataFromFb^.SendSucsess := TRUE;
								OutData[i].InDataFromFb^.SubackQoS := COM.R_BUF.BUFFER[idx + 4];
								OutData[i].step := STEPS_OUT.WAIT_DATA;//can get new data
								OutData[i].TimeOutStarted := FALSE;
								MqttsDoneIo := MqttsDoneIo + 1;
								PaketFound := TRUE;
								//now register callback:
								FOR j := 0 TO CALLBACKS_BUFFER_SIZE - 1 DO
									IF SubscribeCallbacks[j].free THEN
										SubscribeCallbacks[j].free := FALSE;
										SubscribeCallbacks[j].Callback := OutData[i].InDataFromFb^.Callback;
 										SubscribeCallbacks[j].SplitTopic := OutData[i].InDataFromFb^.SplitTopic;
										SubscribeCallbacks[j].ExpectingString := OutData[i].InDataFromFb^.ExpectingString;
										EXIT;
									END_IF
								END_FOR
								IF j = CALLBACKS_BUFFER_SIZE THEN
									//no callback slot free
									OutData[i].InDataFromFb^.CallbackError := TRUE;
								END_IF
								EXIT;
							END_IF
						END_IF
						//
					END_FOR
					IF NOT PaketFound THEN
						CountReceiveSubackUnknown := CountReceiveSubackUnknown + 1;
					END_IF
					idx := idx + SIZE_SUBACK;//only one QoS response expected
				END_IF
			MESSAGETYPE.PUBACK:
				BufferMoveDone := CheckLenghtBuffer(IdxIn:= idx);
				IF NOT BufferMoveDone THEN
					//get Paket ID
					ReceivePaketID := DWORD_TO_WORD(OSCAT_BASIC.DWORD_OF_BYTE(B3:= 0, B2:= 0, 
						B1:= COM.R_BUF.BUFFER[idx + 2],
						B0:= COM.R_BUF.BUFFER[idx + 3]));
					//find Paket
					FOR i := 0 TO MyConstants.QoS_BUFFER_SIZE - 1 DO
						IF OutData[i].step = STEPS_OUT.WAIT_PUBACK THEN //make sure pointer is vailid
							IF OutData[i].InDataFromFb^.PaketId = ReceivePaketID THEN
								OutData[i].InDataFromFb^.SendSucsess := TRUE;
								OutData[i].step := STEPS_OUT.WAIT_DATA;//can get new data
								OutData[i].TimeOutStarted := FALSE;
								MqttsDoneIo := MqttsDoneIo + 1;
								Publishsunacknowledged := Publishsunacknowledged - 1;
								PaketFound := TRUE; 
								EXIT;
							END_IF
						END_IF
						//
					END_FOR
					IF NOT PaketFound THEN
						CountReceivePubackUnknown := CountReceivePubackUnknown + 1;
					END_IF
					idx := idx + SIZE_PUBACK;
				END_IF
			MESSAGETYPE.PUBREC:
				BufferMoveDone := CheckLenghtBuffer(IdxIn:= idx);
				IF NOT BufferMoveDone THEN
					//get Paket ID
					ReceivePaketID := DWORD_TO_WORD(OSCAT_BASIC.DWORD_OF_BYTE(B3:= 0, B2:= 0, 
						B1:= COM.R_BUF.BUFFER[idx + 2],
						B0:= COM.R_BUF.BUFFER[idx + 3]));
					//find Paket
					FOR i := 0 TO MyConstants.QoS_BUFFER_SIZE - 1 DO
						IF OutData[i].step = STEPS_OUT.WAIT_PUBREC THEN //make sure pointer is vailid
							IF OutData[i].InDataFromFb^.PaketId = ReceivePaketID THEN
								IF NOT OutData[i].InDataFromFb^.DUP THEN
									//increase only at first handle 
									PubrelOrderIndexCounter := PubrelOrderIndexCounter + 1;
									OutData[i].PUBRECOrder := PubrelOrderIndexCounter;
								END_IF
								OutData[i].step := STEPS_OUT.SEND_PUBREL;
								OutData[i].TimeOutStarted := FALSE;
								PaketFound := TRUE; 
								EXIT;
							END_IF
						END_IF
						//
					END_FOR
					IF NOT PaketFound THEN
						CountReceivePubrecUnknown := CountReceivePubrecUnknown + 1;
					END_IF
					idx := idx + SIZE_PUBREC;
				END_IF
			MESSAGETYPE.PUBCOMP:
				BufferMoveDone := CheckLenghtBuffer(IdxIn:= idx);
				IF NOT BufferMoveDone THEN
					//get Paket ID
					ReceivePaketID := DWORD_TO_WORD(OSCAT_BASIC.DWORD_OF_BYTE(B3:= 0, B2:= 0, 
						B1:= COM.R_BUF.BUFFER[idx + 2],
						B0:= COM.R_BUF.BUFFER[idx + 3]));
					//find Paket
					FOR i := 0 TO MyConstants.QoS_BUFFER_SIZE - 1 DO
						IF OutData[i].step = STEPS_OUT.WAIT_PUBCOMP THEN //make sure pointer is vailid
							IF OutData[i].InDataFromFb^.PaketId = ReceivePaketID THEN
								OutData[i].InDataFromFb^.SendSucsess := TRUE;
								OutData[i].step := STEPS_OUT.WAIT_DATA;//can get new data
								OutData[i].TimeOutStarted := FALSE;
								MqttsDoneIo := MqttsDoneIo + 1;
								Publishsunacknowledged := Publishsunacknowledged - 1;
								PaketFound := TRUE;
								EXIT;
							END_IF
						END_IF
						//
					END_FOR
					IF NOT PaketFound THEN
						CountReceivePubcompUnknown := CountReceivePubcompUnknown + 1;
					END_IF
					idx := idx + SIZE_PUBCOMP;			
				END_IF
			ELSE
				//unknown paket, reset buffer....
				//standard wants to disconnect....
				{info 'unkown packet, disconnect'}
				LastPaktetForUnkownPaket := HelperLastPaktetForUnkownPaket;
				COM.R_BUF.SIZE := 0;	
				//unknown paket received
				NotKnownPaket := COM.R_BUF.BUFFER[0] AND 16#F0;
				PushError(newError:= ERRORS.UNKNOWN_PAKET_RECEIVED , text:='');
				//alway reset receive!
				COM.MQTT_RCV_STATE := BYTE#0;//receive zurücksetzten
				COM.R_BUF.SIZE := 0;
				CountUnkownPaket := CountUnkownPaket + 1;	
		END_CASE
	UNTIL
		idx >= COM.R_BUF.SIZE OR BufferMoveDone
	END_REPEAT
	IF NOT BufferMoveDone THEN
		COM.R_BUF.SIZE := 0;
	END_IF
	COM.MQTT_RCV_STATE := BYTE#0;//receive zurücksetzten
	
END_IF
                
END_METHOD

METHOD ParseIncomingPublish : UINT
  VAR_INPUT
    MQTT_IN_OUT : POINTER TO MQTT_IN_OUT;
    idx : UINT;  (* pos of paket in buffer *)
    BufferIn : POINTER TO BYTE;  (* give here the buffer were the full packet is... *)
    NetworkBuffer : BOOL;  (* works on network buffer --> need memmove in Output *)
    BufferSize : UDINT;  (* size of buffer, bytes occupied *)
  END_VAR
  VAR
    i : UINT;
    PaketFound : BOOL;
    PaketIndex : UINT;
    FreeSlot : UINT;
    FreeSlotFound : BOOL;
    ReceivePaketID : WORD;
    ReceiveQoSLevel : QoS;
    TopicSize : UINT;
    OutData : BOOL;  (* Output the Data, Tru if Data can be outputted *)
    RemainingLength : REMAINING_LENGTH_RETURN;
    PayloadPosStart : UDINT;
    TopicPosStart : UDINT;
    PayloadSize : UDINT;
    FollowingDataBuffer : ARRAY[0..1] OF BYTE;
    PayloadMoved : BOOL;
  END_VAR
                  ParseIncomingPublish := 0;//if return is zero, buffer move has been done,
CounterPublishReceivedForMonitor := CounterPublishReceivedForMonitor + 1;
GVL_MQTT.ProgNum := PROG_NUM.ParsePublish;
//get remaining length
RemainingLength := GetRemainingLength(BufferIn, pos := idx,BuffSize := BufferSize);
TopicPosStart := RemainingLength.IndexAfterRemainingLength + 2;
ReceiveQoSLevel := SHR(BufferIn[idx] AND 2#110,1);

TopicSize := DWORD_TO_WORD(OSCAT_BASIC.DWORD_OF_BYTE(B3:= 0, B2:= 0,
						 B1:= BufferIn[RemainingLength.IndexAfterRemainingLength],
						 B0:= BufferIn[RemainingLength.IndexAfterRemainingLength+1]));
IF RemainingLength.Error THEN
	//throw away paket on length error
	COM.MQTT_RCV_STATE := BYTE#0;//receive zurücksetzten
	//need to set size to zero, so no further parsing...
	COM.R_BUF.SIZE := 0;
	CountLengthErrors := CountLengthErrors;
	//on standard i MUST diconnect!!!
	DoDisconnect := TRUE;
	PushError(newError:= ERRORS.RECEIVED_PUBLISH_REMAINING_LENGTH_ERROR, text:='');
	
